	//Kapcsolat bontás
	bRobotSocketCloseEnable: BOOL := FALSE;
	RobotSocketClose: FB_SocketClose;
	
	bIsError : BOOL := FALSE;

END_VAR

RobotSocketOpen(
			sSrvNetId:= '', 
			sRemoteHost:= sRobotRemoteHost, 
			nRemotePort:= 2000, 
			bExecute:= bRobotSocketOpenEnable, 
			tTimeout:= T#45S, 
			bBusy=> bConnectBusy, 
			bError=> bConnectError, 
			nErrId=> nConnectErrId, 
			hSocket=> hRobotSocket);
			
RobotSocketSend(
		sSrvNetId:= '', 
		hSocket:= hRobotSocket, 
		cbLen:= uSendByteLen, 
		pSrc:= ADR(baSendByteArray), 
		bExecute:= bRobotSocketSendEnable, 
		tTimeout:= T#5S, 
		bBusy=> bSendBusy, 
		bError=> bSendError, 
		nErrId=> nSendErrId);
		
RobotSocketReceive(
	sSrvNetId:= '', 
	hSocket:= hRobotSocket, 
	cbLen:= 255, 
	pDest:= ADR(baReceivedByteArray), 
	bExecute:= bRobotSocketReceiveEnable, 
	tTimeout:= T#30S, 
	bBusy=> bReceiveBusy, 
	bError=> bReceiveError, 
	nErrId=> nReceiveErrId, 
	nRecBytes=> nRobotReceivedBytesNum);		
		
RobotSocketClose(
	sSrvNetId:= '', 
	hSocket:= hRobotSocket, 
	bExecute:= bRobotSocketCloseEnable, 
	tTimeout:= T#45S, 
	bBusy=> bCloseBusy, 
	bError=> bCloseError, 
	nErrId=> nCloseErrId);

//Kommunikáció nyitás
IF (bRobotCommOpenEnable = TRUE) AND (bRobotCommOpen = FALSE) AND (iState <= 0) THEN
	sRobotResult := '';	
	iState:=1;
ELSE
	bRobotCommOpenEnable := FALSE;
END_IF;

//Parancs küldés
IF (bRobotCommandSend = TRUE) AND (bRobotCommOpen=TRUE) AND(iState <= 0) THEN
	iState:=11;
ELSE
	bRobotCommandSend := FALSE;
END_IF;
//Kommunikáció zárás
IF (bRobotCommCloseEnable = TRUE) AND (bRobotCommOpen = TRUE) AND (iState < 31) THEN
	iState:=31;
ELSE
	bRobotCommCloseEnable := FALSE;
END_IF;




CASE iState OF
	
	1:	//Kommunikáció nyitás
		bRobotSocketOpenEnable:=TRUE;
		iState:=2;
	
	2:
		IF bConnectBusy = TRUE THEN
			iState:=3;
		END_IF
	3:
		IF bConnectBusy = FALSE THEN
			iState:=4;
		END_IF 
		
	4:
		IF bConnectError =FALSE THEN
			//Minden OK
			bRobotCommOpen:=TRUE;
		ELSE
			//HIBA
			bRobotCommOpen:=FALSE;	
		END_IF
		bRobotCommOpenEnable := FALSE;
		bRobotSocketOpenEnable:=FALSE;
		iState:=0;
		
		
	11: //Parancs küldés
		sRobotResult := '';
		nRobotErrId := 0;
		sLRobotCommand := sRobotCommand;
		sRobotSendData := sLRobotCommand;
		baSendByteArray := MAXSTRING_TO_BYTEARR(sRobotSendData);
		uSendByteLen := INT_TO_UDINT(LEN(sRobotSendData));
		MEMSET(ADR(baReceivedByteArray), 0, 256);
		
		iState:=12;
		
	12:
		bRobotSocketSendEnable:=TRUE;
		iState:=13;
		
	13:
		IF bSendBusy = TRUE THEN
			iState:=14;
		END_IF
	14:
		IF bSendBusy = FALSE THEN
			iState:=15;
		END_IF 
		
	15:
		IF bSendError =FALSE THEN
			//Minden OK
			bIsError:= FALSE;
			bRobotSocketReceiveEnable := FALSE;
			iState:=21;
		ELSE
			//HIBA
			bIsError:= TRUE;	
			iState:=0;
		END_IF
		bRobotCommandSend := FALSE;
		bRobotSocketSendEnable:=FALSE;
		
		sRobotCommand:='';		
		sLRobotCommand := '';

		
	21:	//Adatfogadás
		nRobotReceivedBytesNum:=0;
		bRobotSocketReceiveEnable := TRUE;
		iState:=22;
		
	22:
		IF bReceiveBusy = TRUE THEN
			iState:=23;
		END_IF
	23:
		IF bReceiveBusy = FALSE THEN
			iState:=24;
		END_IF 		
	24:
		IF bReceiveError =FALSE THEN
			//Minden OK
			bIsError:= FALSE;
			iState:=25;
		ELSE
			//HIBA
			bIsError:= TRUE;
			iState:=0;	
		END_IF
		bRobotSocketReceiveEnable:=FALSE;
		
	25:
		IF (nRobotReceivedBytesNum <>0) THEN
			sRobotReceived := BYTEARR_TO_MAXSTRING(baReceivedByteArray);
			IF sRobotReceived[0] = 16#30 THEN
				nRobotErrId:= 0;
			ELSE
				nRobotErrId:= 10000;
			END_IF
			GVL.stRobotStatusz:=f_GetRobotState(sRobotReceived);
			sRobotResult:=GVL.stRobotStatusz.sResult;
			iState:=0;
		ELSE
			iState:=21;
		END_IF
		

		
	31:	//Kommunikáció zárás
		bRobotSocketCloseEnable:=TRUE;
		iState:=32;
	
	32:
		IF bCloseBusy = TRUE THEN
			iState:=33;
		END_IF
	33:
		IF bCloseBusy = FALSE THEN
			bRobotSocketCloseEnable:=FALSE;
			iState:=34;
		END_IF 
		
	34:
		IF bCloseError =FALSE THEN
			//Minden OK
			bRobotCommOpen:=FALSE;
		ELSE
			//HIBA
			bRobotCommOpen:=FALSE;	//még át kell gondolni
		END_IF
		bRobotCommCloseEnable := FALSE;
		bRobotSocketCloseEnable:=FALSE;
		iState:=0;
	
END_CASE

END_PROGRAM

// ---- POUs/GENERAL/Helpers/f_GetRobotState.TcPOU
FUNCTION f_GetRobotState : ST_RobotState
VAR_INPUT
	sRobotValasz: STRING;
END_VAR
VAR
	sTemp: STRING;
	sRobotResult: STRING;
	sRobotInput: STRING;
	sRobotCoords: STRING;
	sX: STRING;
	sY: STRING;
	sZ: STRING;
	sU: STRING;
	sHand: STRING;
	nRobotInput: BYTE;
	iDelimiterPos: INT;
END_VAR

sTemp := DELETE(sRobotValasz,1,1);	// Első karakter (0/1) eltávolítása
sTemp := LEFT(sTemp,LEN(sTemp)-2);	// Utolsó két karakter ($R$N) eltávolítása
iDelimiterPos := FIND(sTemp,',');	// Első vessző helye
f_GetRobotState.sResult := LEFT(sTemp,iDelimiterPos-1);	// Vessző előtti szöveg
sTemp := RIGHT(sTemp,LEN(sTemp)-iDelimiterPos); // Vessző utáni szöveg
iDelimiterPos := FIND(sTemp,',');	// Második vessző helye
sRobotInput := LEFT(sTemp,iDelimiterPos-1);	// Vessző előtti szöveg
sTemp := RIGHT(sTemp,LEN(sTemp)-iDelimiterPos); // Vessző utáni szöveg			
iDelimiterPos := FIND(sTemp,',');	// Harmadik vessző helye
sX := LEFT(sTemp,iDelimiterPos-1);	// Vessző előtti szöveg
sTemp := RIGHT(sTemp,LEN(sTemp)-iDelimiterPos); // Vessző utáni szöveg			
iDelimiterPos := FIND(sTemp,',');	// Negyedik vessző helye
sY := LEFT(sTemp,iDelimiterPos-1);	// Vessző előtti szöveg
sTemp := RIGHT(sTemp,LEN(sTemp)-iDelimiterPos); // Vessző utáni szöveg			
iDelimiterPos := FIND(sTemp,',');	// Ötödik vessző helye
sZ := LEFT(sTemp,iDelimiterPos-1); // Vessző előtti szöveg
sTemp := RIGHT(sTemp,LEN(sTemp)-iDelimiterPos); // Vessző utáni szöveg			
iDelimiterPos := FIND(sTemp,',');	// Hatodik vessző helye
sU := LEFT(sTemp,iDelimiterPos-1); // Vessző előtti szöveg			
sHand := RIGHT(sTemp,LEN(sTemp)-iDelimiterPos);	// Vessző utáni szöveg
// nRobotInput bitekre bontása:
nRobotInput := STRING_TO_BYTE(sRobotInput);
f_GetRobotState.bVakuumSzippantoFent:=((nRobotInput AND 1) > 0);
f_GetRobotState.bVakuumSzippantoLent:=((nRobotInput AND 2) > 0);
f_GetRobotState.bCsipeszNyitva:=((nRobotInput AND 4) > 0);
f_GetRobotState.bCsipeszZarva:=((nRobotInput AND 8) > 0);
f_GetRobotState.bVakuumA:=((nRobotInput AND 16) > 0);
f_GetRobotState.bVakuumB:=((nRobotInput AND 32) > 0);
// Robot koordináták:
f_GetRobotState.rX:=STRING_TO_REAL(sX);
f_GetRobotState.rY:=STRING_TO_REAL(sY);
f_GetRobotState.rZ:=STRING_TO_REAL(sZ);
f_GetRobotState.rU:=STRING_TO_REAL(sU);
IF sHand='1' THEN
	sHand:='/R';
ELSIF sHand='2' THEN
	sHand:='/L';
ELSE
	sHand:='/?';
END_IF
f_GetRobotState.sHand:=sHand;

END_FUNCTION

// ---- POUs/JOZSI/Components/HAJLITOK.TcPOU
PROGRAM HAJLITOK
	VAR_INPUT
		s_InCommand : STRING := '';
		s_InCommandParam1 : STRING := '';
		s_InCommandParam2 : STRING := '';
		s_InCommandParam3 : STRING := '';
		s_InCommandParam4 : STRING := '';
		s_InCommandParam5 : STRING := '';
	END_VAR
	VAR_OUTPUT
		n_OutErrId: UINT;
	END_VAR
VAR
	bElohajlitoFelso AT %Q*: BOOL := FALSE;
	bElohajlitoAlso AT %Q*: BOOL := FALSE;
	bVeghajlitoFelso AT %Q*: BOOL := FALSE;
	bVeghajlitoAlso AT %Q*: BOOL := FALSE;
	bElohajlitoFelsoFent AT %I*: BOOL;
	bElohajlitoFelsoLent AT %I*: BOOL;
	bElohajlitoAlsoFent AT %I*: BOOL;
	bElohajlitoAlsoLent AT %I*: BOOL;
	bVeghajlitoFelsoFent AT %I*: BOOL;
	bVeghajlitoFelsoLent AT %I*: BOOL;
	bVeghajlitoAlsoFent AT %I*: BOOL;
	bVeghajlitoAlsoLent AT %I*: BOOL;
	iState : INT := 0;
	s_InLCommand : STRING := '';
	T_Ticker : TON;
	bTickerEnable : BOOL := FALSE;
	tTickerTime : TIME := T#300MS;
	bTickerQ : BOOL := FALSE;
END_VAR

IF HAJLITOK.s_InCommand <>'' AND s_InLCommand = '' THEN
	s_InLCommand := HAJLITOK.s_InCommand;
END_IF
IF s_InLCommand <> '' THEN
	IF iState = 0 AND s_InLCommand = 'ELOHAJLITAS' THEN
		iState := 1;
	END_IF
	IF iState = 0 AND s_InLCommand = 'VEGHAJLITAS' THEN
		iState := 51;
	END_IF
	CASE iState OF 
		1:
			IF (bElohajlitoFelsoFent = TRUE AND bElohajlitoFelsoLent = FALSE
				AND bElohajlitoAlsoFent = FALSE AND bElohajlitoAlsoLent = TRUE) THEN
				n_OutErrId := 0;
				iState := 2;
			ELSIF MAIN.bLevegoOK = FALSE THEN
				n_OutErrId := 5;
			ELSIF bElohajlitoFelsoFent = FALSE THEN
				n_OutErrId := 147;
			ELSIF bElohajlitoFelsoLent = TRUE THEN
				n_OutErrId := 146;
			ELSIF bElohajlitoAlsoFent = TRUE THEN
				n_OutErrId := 151;
			ELSIF bElohajlitoAlsoLent = FALSE THEN
				n_OutErrId := 149;
			END_IF
		2:	// Csak akkor menjen le, ha senki nem nyúlt be
			bElohajlitoFelso := GVL.bFenysorompoNTC;
			iState := 3;
		3:
			IF (bElohajlitoFelsoFent = FALSE AND bElohajlitoFelsoLent = TRUE
				AND bElohajlitoAlsoFent = FALSE AND bElohajlitoAlsoLent = TRUE) THEN
				n_OutErrId := 0;
				iState := 4;
			ELSE
				IF MAIN.bLevegoOK = FALSE THEN
					n_OutErrId := 5;
				ELSIF GVL.bFenysorompoNTC=FALSE THEN
					n_OutErrId := 31;
				ELSIF bElohajlitoFelsoFent = TRUE THEN
					n_OutErrId := 148;
				ELSIF bElohajlitoAlsoFent = TRUE THEN
					n_OutErrId := 152;
				ELSIF bElohajlitoAlsoLent = FALSE THEN
					n_OutErrId := 149;
				END_IF
				bElohajlitoFelso := GVL.bFenysorompoNTC;
			END_IF
		4:	// Csak akkor jöjjön fel, ha senki nem nyúlt be
			bElohajlitoAlso := GVL.bFenysorompoNTC;
			iState := 5;
		5:
			IF (bElohajlitoFelsoFent = FALSE AND bElohajlitoFelsoLent = TRUE
				AND bElohajlitoAlsoFent = TRUE AND bElohajlitoAlsoLent = FALSE) THEN
				n_OutErrId := 0;
				iState := 6;
			ELSE
				IF MAIN.bLevegoOK = FALSE THEN
					n_OutErrId := 5;
				ELSIF GVL.bFenysorompoNTC=FALSE THEN
					n_OutErrId := 31;
				ELSIF bElohajlitoFelsoFent = TRUE THEN
					n_OutErrId := 148;
				ELSIF bElohajlitoAlsoFent = TRUE THEN
					n_OutErrId := 152;
				ELSIF bElohajlitoAlsoLent = FALSE THEN
					n_OutErrId := 149;
				END_IF
				bElohajlitoAlso := GVL.bFenysorompoNTC;
			END_IF
		6:
			IF bTickerEnable = TRUE THEN
				bTickerEnable := FALSE;
			ELSE
				bTickerEnable := TRUE;
				iState := 7;
			END_IF
		7:
			IF bTickerQ = TRUE THEN
				bTickerEnable := FALSE;
				iState := 8;
			END_IF
		8:
			bElohajlitoAlso := FALSE;
			iState := 9;
		9:
			IF (bElohajlitoFelsoFent = FALSE AND bElohajlitoFelsoLent = TRUE
				AND bElohajlitoAlsoFent = FALSE AND bElohajlitoAlsoLent = TRUE) THEN
				n_OutErrId := 0;
				iState := 10;
			ELSIF MAIN.bLevegoOK = FALSE THEN
					n_OutErrId := 5;
			ELSIF bElohajlitoFelsoFent = TRUE THEN
				n_OutErrId := 148;
			ELSIF bElohajlitoFelsoLent = FALSE THEN
				n_OutErrId := 145;
			ELSIF bElohajlitoAlsoFent = TRUE THEN
				n_OutErrId := 152;
			ELSIF bElohajlitoAlsoLent = FALSE THEN
				n_OutErrId := 149;
			END_IF
		10:
			bElohajlitoFelso := FALSE;
			iState := 11;
		11:
			IF (bElohajlitoFelsoFent = TRUE AND bElohajlitoFelsoLent = FALSE
				AND bElohajlitoAlsoFent = FALSE AND bElohajlitoAlsoLent = TRUE) THEN
				iState := 0;
				n_OutErrId := 0;
			ELSIF MAIN.bLevegoOK = FALSE THEN
					n_OutErrId := 5;
			ELSIF bElohajlitoFelsoFent = FALSE THEN
					n_OutErrId := 147;
			ELSIF bElohajlitoFelsoLent = TRUE THEN
					n_OutErrId := 146;
			ELSIF bElohajlitoAlsoFent = TRUE THEN
					n_OutErrId := 152;
			ELSIF bElohajlitoAlsoLent = FALSE THEN
					n_OutErrId := 149;
			END_IF
			
		51:
			IF (bVeghajlitoFelsoFent = TRUE AND bVeghajlitoFelsoLent = FALSE
				AND bVeghajlitoAlsoFent = FALSE AND bVeghajlitoAlsoLent = TRUE) THEN
				n_OutErrId := 0;
				iState := 52;
			ELSIF MAIN.bLevegoOK = FALSE THEN
					n_OutErrId := 5;
			ELSIF bVeghajlitoFelsoFent = FALSE THEN
					n_OutErrId := 163;
			ELSIF bVeghajlitoFelsoLent = TRUE THEN
					n_OutErrId := 162;
			ELSIF bVeghajlitoAlsoFent = TRUE THEN
					n_OutErrId := 166;
			ELSIF bVeghajlitoAlsoLent = FALSE THEN
					n_OutErrId := 167;
			END_IF
		52:
			bVeghajlitoFelso := TRUE;
			iState := 53;
		53:
			IF (bVeghajlitoFelsoFent = FALSE AND bVeghajlitoFelsoLent = TRUE
				AND bVeghajlitoAlsoFent = FALSE AND bVeghajlitoAlsoLent = TRUE) THEN
				n_OutErrId := 0;
				iState := 54;
			ELSIF MAIN.bLevegoOK = FALSE THEN
					n_OutErrId := 5;
			ELSIF bVeghajlitoFelsoFent = TRUE THEN
					n_OutErrId := 164;
			ELSIF bVeghajlitoFelsoLent = FALSE THEN
					n_OutErrId := 161;
			ELSIF bVeghajlitoAlsoFent = TRUE THEN
					n_OutErrId := 166;
			ELSIF bVeghajlitoAlsoLent = FALSE THEN
					n_OutErrId := 167;
			END_IF
		54:
			bVeghajlitoAlso := TRUE;
			iState := 55;
		55:
			IF (bVeghajlitoFelsoFent = FALSE AND bVeghajlitoFelsoLent = TRUE
				AND bVeghajlitoAlsoFent = TRUE AND bVeghajlitoAlsoLent = FALSE) THEN
				n_OutErrId := 0;
				iState := 56;
			ELSIF MAIN.bLevegoOK = FALSE THEN
					n_OutErrId := 5;
			ELSIF bVeghajlitoFelsoFent = TRUE THEN
					n_OutErrId := 164;
			ELSIF bVeghajlitoFelsoLent = FALSE THEN
					n_OutErrId := 161;
			ELSIF bVeghajlitoAlsoFent = FALSE THEN
					n_OutErrId := 165;
			ELSIF bVeghajlitoAlsoLent = TRUE THEN
					n_OutErrId := 168;
			END_IF
		56:
			IF bTickerEnable = TRUE THEN
				bTickerEnable := FALSE;
			ELSE
				bTickerEnable := TRUE;
				iState := 57;
			END_IF
		57:
			IF bTickerQ = TRUE THEN
				bTickerEnable := FALSE;
				iState := 58;
			END_IF
		58:
			bVeghajlitoAlso := FALSE;
			iState := 59;
		59:
			IF (bVeghajlitoFelsoFent = FALSE AND bVeghajlitoFelsoLent = TRUE
				AND bVeghajlitoAlsoFent = FALSE AND bVeghajlitoAlsoLent = TRUE) THEN
				n_OutErrId := 0;
				iState := 60;
			ELSIF MAIN.bLevegoOK = FALSE THEN
				n_OutErrId := 5;
			ELSIF bVeghajlitoFelsoFent = TRUE THEN
				n_OutErrId := 164;
			ELSIF bVeghajlitoFelsoLent = FALSE THEN
				n_OutErrId := 161;
			ELSIF bVeghajlitoAlsoFent = TRUE THEN
				n_OutErrId := 166;
			ELSIF bVeghajlitoAlsoLent = FALSE THEN
				n_OutErrId := 167;
			END_IF
		60:
			bVeghajlitoFelso := FALSE;
			iState := 61;
		61:
			IF (bVeghajlitoFelsoFent = TRUE AND bVeghajlitoFelsoLent = FALSE
				AND bVeghajlitoAlsoFent = FALSE AND bVeghajlitoAlsoLent = TRUE) THEN
				iState := 0;
				n_OutErrId := 0;
			ELSIF MAIN.bLevegoOK = FALSE THEN
				n_OutErrId := 5;
			ELSIF bVeghajlitoFelsoFent = FALSE THEN
				n_OutErrId := 163;
			ELSIF bVeghajlitoFelsoLent = TRUE THEN
				n_OutErrId := 162;
			ELSIF bVeghajlitoAlsoFent = TRUE THEN
				n_OutErrId := 166;
			ELSIF bVeghajlitoAlsoLent = FALSE THEN
				n_OutErrId := 167;
			END_IF
			
	END_CASE
	IF iState = 0 THEN
		HAJLITOK.s_InCommand := '';
		s_InLCommand := '';
	END_IF
END_IF

T_Ticker(IN:= bTickerEnable, PT:= tTickerTime, Q=> bTickerQ, ET=> );

END_PROGRAM

// ---- POUs/PISTI/Components/PISTITENGELY.TcPOU
PROGRAM PISTITENGELY
VAR
	PistiHome: MC_Home;
	bPistiHomeEnable: BOOL := FALSE;
	bAxisBusy : BOOL := FALSE;
	bAxisActive: BOOL := FALSE;
	bAxisAborted: BOOL := FALSE;
	bAxisError: BOOL := FALSE;
	nAxisErrorID: UDINT;
	bAxisStopDone: BOOL := FALSE;
	bPistiHomeSwitch AT %I*: BOOL;
	fbPistiTengelyStop: MC_Stop;
	fbPistitengelyServo: MC_Power;
	bPistiPosSwitch : BOOL := TRUE;
	bPistiTengelySzabad : BOOL;
	bOperational AT %I*: BOOL;
	bHomeReady : BOOL := FALSE;
	nAxisStatus AT %I*: UINT;
	bAxisReady : BOOL;
	bAxisOn : BOOL;
	
	//HOME
	bAxisHomeDone: BOOL;
	bAxisHomeBusy: BOOL;
	bAxisHomeActive: BOOL;
	bAxisHomeAborted: BOOL;
	bAxisHomeError: BOOL;
	nAxisHomeErrorID: UDINT;
	
	//MOVE
	bAxisMoveDone: BOOL;
	bAxisMoveBusy: BOOL;
	bAxisMoveActive: BOOL;
	bAxisMoveAborted: BOOL;
	bAxisMoveError: BOOL;
	nAxisMoveErrorID: UDINT;
	
	//COMMAND
	bAxisCommandDone: BOOL;
	bAxisCommandBusy: BOOL;
	bAxisCommandActive: BOOL;
	bAxisCommandAborted: BOOL;
	bAxisCommandError: BOOL;
	nAxisCommandErrorID: UDINT;
	
	
	fbPistitengelyJOG: MC_Jog;
	bPistiJOGPlus : BOOL := FALSE;
	bPistiJOGMinus : BOOL := FALSE;
	fbPistitengelyReset: MC_Reset;
	bPistiReset: BOOL;
	nPistiErrorCode AT %I*: UDINT;
	lrPistiActPos AT %I*: LREAL;
	fbPistiMoveAbolute: MC_MoveAbsolute;
	
	//Pozicioknak
//	lrSzervizbox : LREAL := -5;
//	lrHegesztoPosition1 : LREAL := -398.3;
//	lrHegesztoPosition2 : LREAL := -404.3;
//	lrRobotpakolasPosition : LREAL := -617.8125;
//	lrKodolvasasPosition: LREAL := -841.54;
//	lrKappePosition : LREAL := -837.227;
//	lrVegmeroPosition : LREAL := -1054.776;
	bPistiTengelySzabad_TON: TON;
END_VAR
VAR_INPUT
	lrPistiPosition : LREAL := 0;
	sPistiAxisCommand: STRING := '';
END_VAR
VAR_OUTPUT
	n_OutErrId: UINT;
END_VAR

//bPistiTengelySzabad := GVL.bTempPistiInputs1[3] AND GVL.bTempPistiInputs2[6]
bPistiTengelySzabad := GVL.bHegeszto3Fent AND GVL.bKappepresFent
						AND VEGMERO.bMerotukBent AND (HIMBA.bHimba_hatul AND NOT HIMBA.bHimba_elol) AND bOperational
//						AND ((GVL.stRobotStatusz.rX<-1.0) OR (GVL.stRobotStatusz.rZ>-111.0))
						AND f_RobotPtTengelytolTavol()
						AND (GVL.bFenysorompoPt
							OR (sPistiAxisCommand='HOME')
							OR (PISTITENGELY.lrPistiActPos>-10)
							OR (PISTITENGELY.lrPistiActPos<-500))
						AND NOT GVL.bBiztonsagiFold AND GVL.bBiztonsagiTap;
bPistiTengelySzabad_TON(IN:=bPistiTengelySzabad, PT:=T#100MS);
IF bPistiTengelySzabad_TON.Q=FALSE THEN
	IF MAIN.bLevegoOK=FALSE THEN
		n_OutErrId:=5;
	ELSIF GVL.bHegeszto3Fent=FALSE THEN
		n_OutErrId:=71;
	ELSIF GVL.bKappepresFent=FALSE THEN
		n_OutErrId:=109;
	ELSIF VEGMERO.bMerotukBent=FALSE THEN
		n_OutErrId:=87;
	ELSIF HIMBA.bHimba_hatul=FALSE OR HIMBA.bHimba_elol=TRUE THEN
		n_OutErrId:=339;
	ELSIF bOperational=FALSE THEN
		n_OutErrId:=195;
//	ELSIF NOT ((GVL.stRobotStatusz.rX<-1.0) OR (GVL.stRobotStatusz.rZ>-111.0)) THEN
	ELSIF NOT f_RobotPtTengelytolTavol() THEN
		n_OutErrId:=302;
	ELSIF (GVL.bFenysorompoPt=FALSE) THEN
		n_OutErrId:=29;
	ELSIF GVL.bBiztonsagiFold=TRUE THEN
		n_OutErrId:=42;
	ELSIF GVL.bBiztonsagiTap=FALSE THEN
		n_OutErrId:=43;
	END_IF
ELSE
	n_OutErrId := 0;
END_IF
bAxisReady:=nAxisStatus MOD 2 = 1;
bAxisOn:=nAxisStatus/2 MOD 2 = 1;
fbPistiTengelyStop(
	Axis:= GVL.axisPistiTengely, 
	Execute:= (NOT((GVL.bPistiPosSwitch OR sPistiAxisCommand='HOME') AND GVL.bPistiNegSwitch AND bPistiTengelySzabad_TON.Q)
				OR sPistiAxisCommand='STOP'), 
	Deceleration:= , 
	Jerk:= , 
	Options:= , 
	Done=> PISTITENGELY.bAxisStopDone, 
	Busy=> bAxisBusy, 
	Active=> bAxisActive, 
	CommandAborted=> bAxisAborted, 
	Error=> bAxisError, 
	ErrorID=> nAxisErrorID);
IF (sPistiAxisCommand='STOP') AND PISTITENGELY.bAxisStopDone AND NOT bAxisError THEN
	sPistiAxisCommand := '';
END_IF
IF NOT(GVL.bPistiPosSwitch OR sPistiAxisCommand='HOME') OR NOT(GVL.bPistiNegSwitch) THEN
	GVL.bPistiServo := FALSE;
	sPistiAxisCommand:='';
END_IF
fbPistitengelyServo(
	Axis:= GVL.axisPistiTengely, 
	Enable:= GVL.bPistiServo, 
	Enable_Positive:= (GVL.bPistiPosSwitch OR sPistiAxisCommand='HOME'), 
	Enable_Negative:= GVL.bPistiNegSwitch, 
	Override:= 100, 
	BufferMode:= , 
	Options:= , 
	Status=> , 
	Busy=> , 
	Active=> , 
	Error=> , 
	ErrorID=> );
	
	//Home
PistiHome(
	Axis:= GVL.axisPistiTengely, 
	Execute:= sPistiAxisCommand='HOME' AND bPistiTengelySzabad_TON.Q, 
	Position:= DEFAULT_HOME_POSITION, 
	HomingMode:= MC_DefaultHoming, 
	BufferMode:= , 
	Options:= , 
	bCalibrationCam:= NOT(bPistiHomeSwitch), 
	Done=> bAxisHomeDone, 
	Busy=> bAxisHomeBusy, 
	Active=> bAxisHomeActive, 
	CommandAborted=> bAxisHomeAborted, 
	Error=> bAxisHomeError, 
	ErrorID=> nAxisHomeErrorID);
	//Lefutás ellenőrzése
IF (bAxisHomeDone AND NOT(bAxisHomeBusy OR bAxisHomeActive OR bAxisHomeAborted OR bAxisHomeError)) THEN
	lrPistiPosition:=GVL.lrPtSzervizbox;
	sPistiAxisCommand := 'MOVE';
	bHomeReady:=TRUE;
END_IF
	
	//Move
fbPistiMoveAbolute(
	Axis:= GVL.axisPistiTengely, 
	Execute:= sPistiAxisCommand='MOVE' AND bPistiTengelySzabad_TON.Q AND bHomeReady, 
	Position:= lrPistiPosition, // -1060...0
	Velocity:= 800, 
	Acceleration:= 0, 
	Deceleration:= 0, 
	Jerk:= 0, 
	BufferMode:= , 
	Options:= , 
	Done=> bAxisMoveDone, 
	Busy=> bAxisMoveBusy, 
	Active=> bAxisMoveActive, 
	CommandAborted=> bAxisMoveAborted, 
	Error=> bAxisMoveError, 
	ErrorID=> nAxisMoveErrorID);
	//Lefutás ellenőrzése
IF (bAxisMoveDone AND NOT(bAxisMoveBusy OR bAxisMoveActive OR bAxisMoveAborted OR bAxisMoveError)) THEN
	sPistiAxisCommand := '';
END_IF
	
	//JOG
	fbPistitengelyJOG(
	Axis:= GVL.axisPistiTengely, 
	JogForward:= bPistiJOGPlus AND bPistiTengelySzabad_TON.Q, 
	JogBackwards:= bPistiJOGMinus AND bPistiTengelySzabad_TON.Q, 
	Mode:= MC_JOGMODE_STANDARD_SLOW , 
	Position:= , 
	Velocity:= 100, 
	Acceleration:= 0, 
	Deceleration:= 0, 
	Jerk:= 0, 
	Done=> bAxisCommandDone, 
	Busy=> bAxisCommandBusy, 
	Active=> bAxisCommandActive, 
	CommandAborted=> bAxisCommandAborted, 
	Error=> bAxisCommandError, 
	ErrorID=> nAxisCommandErrorID);
	
	//RESET ERROR
	fbPistitengelyReset(
	Axis:= GVL.axisPistiTengely, 
	Execute:= bPistiReset, 
	Done=> bAxisCommandDone, 
	Busy=> bAxisCommandBusy, 
	Error=> bAxisCommandError, 
	ErrorID=> nAxisCommandErrorID);
	
	//Ha nem szabad futtatni
//	IF(NOT(bPistiTengelySzabad)) THEN
//		sPistiAxisCommand:='!INTERRUPTED';
//	END_IF

END_PROGRAM

// ---- POUs/PISTI/Components/HIMBA.TcPOU
PROGRAM HIMBA
VAR_INPUT
	s_InCommand : STRING := '';
	s_InCommandParam1 : STRING := '';
	s_InCommandParam2 : STRING := '';
	s_InCommandParam3 : STRING := '';
	s_InCommandParam4 : STRING := '';
	s_InCommandParam5 : STRING := '';
END_VAR
VAR_OUTPUT
	n_OutErrId: UINT;
END_VAR
VAR
	bHimba_hatul AT %I*: BOOL; //6
	bHimba_elol AT %I*: BOOL; //7
	bHimba_szenzor AT %I*: BOOL; //Bemenetek2 10
	bHimba AT %Q*: BOOL := 0; //Szelep11
	iState: INT;
	WAIT: TON;
	bStartWait: BOOL := FALSE;
	bIdoLejart: BOOL := FALSE;
	tDelay: TIME := T#2000MS;
END_VAR

IF (iState=0) AND (HIMBA.s_InCommand='START') THEN
	iState:=1;
ELSIF (iState<20) AND (HIMBA.s_InCommand='RESET') THEN
	iState:=20;
END_IF

	IF iState<>0 THEN
		CASE iState OF
		// Himba kitolása
		1:	GVL.bHimbaOK:=FALSE;
			HIMBA.bHimba:=TRUE;
			iState:=2;
		// Ha megérkezett a Himba, várunk a megnyugvásra
		2:	IF (HIMBA.bHimba_elol=TRUE) AND (HIMBA.bHimba_hatul=FALSE) THEN
				tDelay:=T#600MS;
				bStartWait:=TRUE;
				n_OutErrId:=0;
				iState:=3;
			ELSE
				n_OutErrId:=338;
			END_IF
		// Ha lejárt a várakozási idő kiértékeljük az érzékelő jelét
		3:	IF (bIdoLejart=TRUE) THEN
				bStartWait:=FALSE;
				IF (HIMBA.bHimba_szenzor=TRUE) THEN
					GVL.bHimbaOK:=TRUE;
				ELSE
					GVL.bHimbaOK:=FALSE;
				END_IF
				iState:=4;
			END_IF
		// Himba visszahúzása
		4:	HIMBA.bHimba:=FALSE;
			iState:=5;
		// Ha visszatért a himba, várunk a megnyugvásra
		5: IF (HIMBA.bHimba_hatul=TRUE) AND (HIMBA.bHimba_elol=FALSE) THEN
				tDelay:=T#300MS;
				bStartWait:=TRUE;
				n_OutErrId:=0;
				iState:=6;
			ELSE
				n_OutErrId:=339;
			END_IF
		// Ha lejárt az idő, vége a folyamatnak
		6:	IF (bIdoLejart=TRUE) THEN
				bStartWait:=FALSE;
				iState:=0;
				HIMBA.s_InCommand:='';
			END_IF

		// Reset: húzza vissza a himbát!
		20:	bStartWait:=FALSE;
			GVL.bHimbaOK:=FALSE;
			HIMBA.bHimba:=FALSE;
			iState:=21;				
		// Ha visszatért a himba, várunk a megnyugvásra
		21:	IF (HIMBA.bHimba_hatul=TRUE) AND (HIMBA.bHimba_elol=FALSE) THEN
				tDelay:=T#300MS;
				bStartWait:=TRUE;
				n_OutErrId:=0;
				iState:=22;
			ELSE
				n_OutErrId:=339;
			END_IF
		// Ha lejárt az idő, vége a folyamatnak
		22:	IF (bIdoLejart=TRUE) THEN
				bStartWait:=FALSE;
				iState:=0;
				HIMBA.s_InCommand:='';
			END_IF
		END_CASE
	END_IF	

WAIT(IN:=bStartWait,PT:=tDelay,Q=>bIdoLejart,ET=>);

END_PROGRAM

// ---- POUs/GENERAL/Helpers/f_RobotPtTengelytolTavol.TcPOU
FUNCTION f_RobotPtTengelytolTavol : BOOL

f_RobotPtTengelytolTavol:=(GVL.stRobotStatusz.rX<-1.0) OR (GVL.stRobotStatusz.rZ>-111.0);

END_FUNCTION

// ---- POUs/PISTI/Components/KAPPE.TcPOU
PROGRAM KAPPE
VAR_INPUT
	s_InCommand : STRING := '';
	s_InCommandParam1 : STRING := '';
	s_InCommandParam2 : STRING := '';
	s_InCommandParam3 : STRING := '';
	s_InCommandParam4 : STRING := '';
	s_InCommandParam5 : STRING := '';
END_VAR
VAR_OUTPUT
	n_OutErrId: UINT;
END_VAR
VAR
	bKappeFelLe AT %Q*: BOOL := 0;
	bKappeBalFelLe AT %Q*: BOOL := 0;
	bKappeJobbFelLe AT %Q*: BOOL := 0;
	bKappeNincsLegalul AT %I*: BOOL;
	bKappeFent AT %I*: BOOL;
	bKappeBalFent AT %I*: BOOL;
	bKappeBalLent AT %I*: BOOL;
	bKappeJobbFent AT %I*: BOOL;
	bKappeJobbLent AT %I*: BOOL;
	iState: INT;
	WAIT: TON;
	bStartWait: BOOL := FALSE;
	bIdoLejart: BOOL := FALSE;
	tDelay: TIME := T#2000MS;
END_VAR

IF (iState=0) AND (KAPPE.s_InCommand='START') THEN
	iState:=1;
ELSIF (iState<20) AND (KAPPE.s_InCommand='RESET') THEN
	iState:=20;
END_IF
	IF iState<>0 THEN
		CASE iState OF
		// Kappe fej leeresztése
		1:	KAPPE.bKappeFelLe:=TRUE;
			iState:=2;
		// Ha leérkezett a Kappe fej, akkor várakozik a nyugvópontra
		2:	IF (GVL.bKappepresNincsLegalul=FALSE) THEN
				tDelay:=T#200MS;
				bStartWait:=TRUE;
				n_OutErrId := 0;
				iState:=3;
			ELSE
				IF MAIN.bLevegoOK=FALSE THEN
					n_OutErrId:=5;
				ELSE
					n_OutErrId:=94;
				END_IF
			END_IF
		// Ha lejárt a várakozási idő és a kappézó ujjak ki vannak nyitva,
		// akkor zárja be az ujjakat!
		3:	IF (bIdoLejart=TRUE) AND (KAPPE.bKappeBalFent=TRUE) 
				AND (KAPPE.bKappeBalLent=FALSE) AND (KAPPE.bKappeJobbFent=TRUE)
				AND (KAPPE.bKappeJobbLent=FALSE) THEN
				bStartWait:=FALSE;
				KAPPE.bKappeBalFelLe:=TRUE;
				KAPPE.bKappeJobbFelLe:=TRUE;
				n_OutErrId := 0;
				iState:=4;
			ELSIF MAIN.bLevegoOK=FALSE THEN
				n_OutErrId:=5;
			ELSIF (KAPPE.bKappeBalFent=FALSE) THEN
				n_OutErrId:=101;
			ELSIF (KAPPE.bKappeBalLent=TRUE) THEN
				n_OutErrId:=104;
			ELSIF (KAPPE.bKappeJobbFent=FALSE) THEN
				n_OutErrId:=99;
			ELSIF (KAPPE.bKappeJobbLent=TRUE) THEN
				n_OutErrId:=98;
			END_IF
		// Ha megnyomta a Kappét, várjon egy kicsit!
		4:	IF (KAPPE.bKappeBalFent=FALSE) AND (KAPPE.bKappeBalLent=TRUE)
				AND (KAPPE.bKappeJobbFent=FALSE) AND (KAPPE.bKappeJobbLent=TRUE) THEN
				tDelay:=T#1000MS;
				bStartWait:=TRUE;
				n_OutErrId := 0;
				iState:=5;
			ELSIF MAIN.bLevegoOK=FALSE THEN
				n_OutErrId:=5;
			ELSIF (KAPPE.bKappeBalFent=TRUE) THEN
				n_OutErrId:=102;
			ELSIF (KAPPE.bKappeBalLent=FALSE) THEN
				n_OutErrId:=103;
			ELSIF (KAPPE.bKappeJobbFent=TRUE) THEN
				n_OutErrId:=100;
			ELSIF (KAPPE.bKappeJobbLent=FALSE) THEN
				n_OutErrId:=97;
			END_IF
		// A várakozás után nyissa ki a kappézó ujjakat!
		5:	IF (bIdoLejart=TRUE) THEN
				bStartWait:=FALSE;
				KAPPE.bKappeBalFelLe:=FALSE;
				KAPPE.bKappeJobbFelLe:=FALSE;
				iState:=6;				
			END_IF
		// Ha kinyíltak a kappézó ujjak, akkor Kappe fej fel
		6:	IF (KAPPE.bKappeBalFent=TRUE) AND (KAPPE.bKappeBalLent=FALSE)
				AND (KAPPE.bKappeJobbFent=TRUE) AND (KAPPE.bKappeJobbLent=FALSE) THEN
				KAPPE.bKappeFelLe:=FALSE;
				tDelay:=T#2000MS;
				bStartWait:=TRUE;
				n_OutErrId := 0;
				iState:=7;
			ELSIF MAIN.bLevegoOK=FALSE THEN
				n_OutErrId:=5;
			ELSIF (KAPPE.bKappeBalFent=FALSE) THEN
				n_OutErrId:=101;
			ELSIF (KAPPE.bKappeBalLent=TRUE) THEN
				n_OutErrId:=104;
			ELSIF (KAPPE.bKappeJobbFent=FALSE) THEN
				n_OutErrId:=99;
			ELSIF (KAPPE.bKappeJobbLent=TRUE) THEN				
				n_OutErrId:=98;
			END_IF
		// Ha felemelkedett a Kappe fej, akkor vége a folyamatnak
		7:	IF (GVL.bKappePresFent=TRUE) THEN
				bStartWait:=FALSE;				
				n_OutErrId:=0;
				iState:=0;
				KAPPE.s_InCommand:='';
			ELSIF MAIN.bLevegoOK=FALSE THEN
				n_OutErrId:=5;
			ELSIF (GVL.bKappePresFent=FALSE) THEN
				n_OutErrId:=205;
			END_IF
		// Reset: nyissa ki a kappézó ujjakat!
		20:	bStartWait:=FALSE;
			KAPPE.bKappeBalFelLe:=FALSE;
			KAPPE.bKappeJobbFelLe:=FALSE;
			iState:=21;				
		// Ha kinyíltak a kappézó ujjak, akkor Kappe fej fel
		21:	IF (KAPPE.bKappeBalFent=TRUE) AND (KAPPE.bKappeBalLent=FALSE)
				AND (KAPPE.bKappeJobbFent=TRUE) AND (KAPPE.bKappeJobbLent=FALSE) THEN
				KAPPE.bKappeFelLe:=FALSE;
				tDelay:=T#2000MS;
				bStartWait:=TRUE;
				n_OutErrId := 0;
				iState:=22;
			ELSIF MAIN.bLevegoOK=FALSE THEN
				n_OutErrId:=5;
			ELSIF (KAPPE.bKappeBalFent=FALSE) THEN
				n_OutErrId:=101;
			ELSIF (KAPPE.bKappeBalLent=TRUE) THEN
				n_OutErrId:=104;
			ELSIF (KAPPE.bKappeJobbFent=FALSE) THEN
				n_OutErrId:=99;
			ELSIF (KAPPE.bKappeJobbLent=TRUE) THEN				
				n_OutErrId:=98;
			END_IF
		// Ha felemelkedett a Kappe fej, akkor vége a folyamatnak
		22:	IF (GVL.bKappePresFent=TRUE) THEN
				bStartWait:=FALSE;				
				n_OutErrId:=0;
				iState:=0;
				KAPPE.s_InCommand:='';
			ELSIF MAIN.bLevegoOK=FALSE THEN
				n_OutErrId:=5;
			ELSIF (GVL.bKappePresFent=FALSE) THEN
				n_OutErrId:=205;
			END_IF
		END_CASE
	END_IF	
WAIT(IN:=bStartWait,PT:=tDelay,Q=>bIdoLejart,ET=>);

END_PROGRAM

// ---- POUs/GENERAL/Components/TERMEKVALTAS.TcPOU
PROGRAM TERMEKVALTAS
VAR_INPUT
	iState: INT := 1;
	bStart: BOOL := FALSE;
END_VAR
VAR_OUTPUT
	bOK: BOOL := FALSE;
	bBusy: BOOL := FALSE;
END_VAR

CASE iState OF
	1:
		IF (GVL.iPreviousSelectedProductType<>GVL.iSelectedProductType) OR
			(bStart=TRUE) THEN
			bOK:=FALSE;
			bBusy:=TRUE;
			iState:=2;
			GVL.iCurrentProductType:=-3; // Kérje az etalonokat!
		END_IF
	2:
		IF NOT(GVL.iSelectedProductType=8) THEN
			IF(GVL.iSelectedProductType<8) THEN
				Laser.s_InCommand:='SETJOB_637';
			ELSE
				CASE GVL.iSelectedProductType OF
					9, 11, 13, 15: Laser.s_InCommand:='SETJOB_745900';
					10, 12, 14, 16: Laser.s_InCommand:='SETJOB_745910';
				END_CASE
(*			ELSIF GVL.iSelectedProductType=9 THEN
				Laser.s_InCommand:='SETJOB_745900';
			ELSIF GVL.iSelectedProductType=10 THEN
				Laser.s_InCommand:='SETJOB_745910';*)
			END_IF;
			GVL.bKameraBe := TRUE;
			GVL.bHajlitasBe := TRUE;
			GVL.bHegesztes1Be := TRUE;
			GVL.bHegesztes2Be := TRUE;
			GVL.bHegesztes3Be := TRUE;
			GVL.bHegesztes4Be := TRUE;
			GVL.bHegesztes5Be := TRUE;
			GVL.bKameraVegBe := FALSE;
			GVL.bHegesztes6Be := TRUE;
			GVL.bHegesztes7Be := TRUE;
			GVL.bPtKameraBe := TRUE;
			GVL.bRobotKappeBe := FALSE;
			GVL.bKappeBe := TRUE;
			GVL.bMeresBe := TRUE;
			IF (GVL.iSelectedProductType>8) THEN
				GVL.bHimbaBe := TRUE;
			ELSE
				GVL.bHimbaBe := FALSE;
			END_IF
			GVL.bJelolesBe := TRUE;	
			iState:=3;
		ELSIF GVL.iSelectedProductType=8 THEN
			Laser.s_InCommand:='SETJOB_521';
			GVL.bKameraBe := FALSE;
			GVL.bHajlitasBe := FALSE;
			GVL.bHegesztes1Be := FALSE;
			GVL.bHegesztes2Be := FALSE;
			GVL.bHegesztes3Be := FALSE;
			GVL.bHegesztes4Be := FALSE;
			GVL.bHegesztes5Be := FALSE;
			GVL.bKameraVegBe := FALSE;
			GVL.bHegesztes6Be := FALSE;
			GVL.bHegesztes7Be := FALSE;
			GVL.bPtKameraBe := FALSE;
			GVL.bRobotKappeBe := FALSE;
			GVL.bKappeBe := FALSE;
			GVL.bMeresBe := FALSE;
			GVL.bHimbaBe := FALSE;
			GVL.bJelolesBe := TRUE;	
			iState:=4;
		ELSE
			iState:=1;
			GVL.iSelectedProductType:=GVL.iPreviousSelectedProductType;
			bOK:=FALSE;
			bBusy:=FALSE;
		END_IF
	3:
		IF Laser.s_InCommand='' THEN
			Laser.s_InCommand:='SETTYPE';
			iState:=4;
		END_IF
	4:
		IF Laser.s_InCommand='' THEN
			iState:=1;
			bOK:=TRUE;
			bBusy:=FALSE;
			bStart:=FALSE;
			GVL.iPreviousSelectedProductType:=GVL.iSelectedProductType;
		ELSIF Laser.s_InCommand<>'SETTYPE' THEN
			iState:=1;
			bOK:=FALSE;
			bBusy:=FALSE;
			bStart:=FALSE;
			GVL.iPreviousSelectedProductType:=GVL.iSelectedProductType;
		END_IF	
END_CASE

END_PROGRAM

// ---- POUs/PISTI/Components/ZEBRASCANNER.TcPOU
PROGRAM ZEBRASCANNER
VAR
	iState: INT := 0;
	// I/O variables for a PC COM PORT
	InputBuffer AT %I*: PcComInData;
	OutputBuffer AT %Q*: PcComOutData;
	TxBufferPcCom: COMbuffer;
	RxBufferPcCom: COMbuffer;

	// Serial line control for virtual COM port
	fbPCComCtrl: SerialLineControlADS;
	bConnect: BOOL := TRUE;
//	stSerialCfg: ComSerialConfig := (ComPort := 5, DTR := COMDTRCTRL_T.DTR_CTRL_DISABLE, RTS := COMRTSCTRL_T.RTS_CTRL_ENABLE);
	stSerialCfg: ComSerialConfig := (ComPort := 7, Baudrate:=115200, Parity:=PARITY_EVEN, DTR := COMDTRCTRL_T.DTR_CTRL_DISABLE, RTS := COMRTSCTRL_T.RTS_CTRL_ENABLE);
	stSerialCfgZebra: ComSerialConfig := (ComPort := 5, DTR := COMDTRCTRL_T.DTR_CTRL_DISABLE, RTS := COMRTSCTRL_T.RTS_CTRL_ENABLE);
	stSerialCfgKeyence: ComSerialConfig := (ComPort := 7, Baudrate:=115200, Parity:=PARITY_EVEN, DTR := COMDTRCTRL_T.DTR_CTRL_DISABLE, RTS := COMRTSCTRL_T.RTS_CTRL_ENABLE);
	bPortOpened: BOOL;
	bPcComCtrlError: BOOL;
	ePcComCtrlErrorId: UDINT;
	bPCComCtrlBusy: BOOL;
	uiTxBufferCount: UDINT;
	uiRxBufferCount: UDINT;
	
//	fbPCComCtrl2: SerialLineControl;
	
	// Receiving
	ZebraReceiveString: ReceiveString;
	bReset: BOOL;
	sReceivedString: STRING;
	bStringReceived: BOOL;
	bBusy: BOOL;
	cetError: ComError_t;
	bRxTimeout: BOOL;
	
	// Sending
	ZebraSendString: SendString;	
	sStringToSend: STRING;
	bSendBusy: BOOL;
	eSendError: ComError_t;
	sStartScanning: STRING := '$04$E4$04$00$00$14';
	iSendDataLength: UDINT := 6;
	
	// Sending bytes
	nSentBytes: DINT;
	ZebraSendData: SendData;
	
	// Receiving bytes
	nReceivedBytes: DINT;
	baReceivedBytes: ARRAY[0..255] OF BYTE;
	ZebraReceiveBytes: ReceiveByte;
	ReceiveString255: ReceiveString255;
	ClearComBuffer: ClearComBuffer;
	sExpectedString: T_MaxString;
	
	GetTime: NT_GetTime;
	bStartGetTime: BOOL;
	bGetTimeBusy: BOOL;
	bGetTimeError: BOOL;
	nGetTimeError: UDINT;
	sYear: STRING;
	sMonth: STRING;
	sDay: STRING;
	tstDateTime: TIMESTRUCT;
	sTypeCode: STRING;
	Timer: TON;
	bStart: BOOL;
	tTimeOut: TIME := T#3S;
	bTimeOut: BOOL;
	tElapsedTime: TIME;
	bKeyence: BOOL;
	iInd: INT;
END_VAR

VAR_INPUT
	bStartSend: BOOL;	
END_VAR

VAR_OUTPUT
	sReceivedString255: T_MaxString;
	nReceivedStringLength: DINT;
	bReadReady: BOOL := FALSE;	
END_VAR

(*VAR_IN_OUT
	sExpectedString: T_MaxString;
END_VAR*)

VAR CONSTANT
	baStartScanning: ARRAY[0..5] OF BYTE := [16#4, 16#E4, 16#4, 16#0, 16#FF, 16#14];
	baStartScanningKeyence: ARRAY[0..3] OF BYTE := [16#4C, 16#4F, 16#4E, 16#0D];
END_VAR

fbPCComCtrl(
	Connect:=bConnect,
	SerialCfg:=stSerialCfg,
	NetId:='',
	Timeout:=T#2s,
	PortOpened=>bPortOpened,
	Error=>bPCComCtrlError,
	ErrorId=>ePCComCtrlErrorId,
	Busy=>bPCComCtrlBusy,
	TxBufCount=>uiTxBufferCount,
	RxBufCount=>uiRxBufferCount,
	TxBuffer:=TxBufferPcCom,
	RxBuffer:=RxBufferPcCom);

REPEAT
	ZebraReceiveBytes(Rxbuffer:=RxBufferPcCom);
	IF ZebraReceiveBytes.ByteReceived THEN
		IF nReceivedBytes=0 THEN
			FOR nReceivedBytes:=0 TO 255 DO
				baReceivedBytes[nReceivedBytes]:=0;
			END_FOR
			nReceivedBytes:=0;
		END_IF
		baReceivedBytes[nReceivedBytes]:=ZebraReceiveBytes.ReceivedByte;
		nReceivedBytes:=nReceivedBytes+1;
	END_IF
UNTIL NOT ZebraReceiveBytes.ByteReceived
END_REPEAT;

(*REPEAT
	ReceiveString255(Suffix:='$R',
					Timeout:=T#10MS,
					RxTimeout=>bRxTimeout, StringReceived=>bStringReceived,
					ReceivedString:=sReceivedString255,
					Rxbuffer:=RxBufferPcCom);
UNTIL bStringReceived OR bRxTimeout
END_REPEAT;*)

(*IF bStringReceived THEN
	iState:=1;
END_IF*)

IF nReceivedBytes>0 THEN
	FOR iInd:=0 TO 255 DO
		baReceivedBytes[iInd]:=0;
	END_FOR
	IF (GVL.iSelectedProductType<8) THEN // Ha 6379XX termék
		FOR iInd:=0 TO 26 DO
			baReceivedBytes[iInd]:=RxBufferPcCom.Buffer[iInd];
		END_FOR
	ELSE // Ha 521950 vagy 7459XX termék: 1 karakterrel kevesebb
		FOR iInd:=0 TO 25 DO
			baReceivedBytes[iInd]:=RxBufferPcCom.Buffer[iInd];
		END_FOR
	END_IF
	sReceivedString255:=BYTEARR_TO_MAXSTRING(baReceivedBytes);
	IF LEFT(sReceivedString255,5)='ERROR' THEN
		sReceivedString255:='ERROR';
	END_IF
	nReceivedStringLength:=LEN(sReceivedString255);
	IF nReceivedStringLength>20 THEN
		iState:=1;
	END_IF
	nReceivedBytes:=0;
END_IF

(*ZebraReceiveString(
	Prefix:='',
	Suffix:='',
	Timeout:=T#1S,
	Reset:=bReset,
	StringReceived=>bStringReceived,
	Busy=>bBusy,
	Error=>cetError,
	RxTimeout=>bRxTimeout,
	ReceivedString:=sReceivedString,
	Rxbuffer:=RxBufferPcCom);*)

IF iState=0 AND (bStartSend=TRUE OR bSendBusy=TRUE) THEN
	IF bStartSend=TRUE THEN
//		sStringToSend:=sStartScanning;
		sReceivedString255:='';
		nReceivedStringLength:=0;
		bReadReady:=FALSE;
		GVL.bMarkingOK:=FALSE;
		GVL.iMarkingQ:=0;
		bStart:=TRUE;
	END_IF
(*	IF NOT bKeyence THEN
		ZebraSendData(
			pSendData:=ADR(baStartScanning),
			Length:=6,
			Busy=>bSendBusy,
			Error=>eSendError,
			TXbuffer:=TxBufferPcCom);
	ELSE
		ZebraSendData(
			pSendData:=ADR(baStartScanningKeyence),
			Length:=4,
			Busy=>bSendBusy,
			Error=>eSendError,
			TXbuffer:=TxBufferPcCom);
	END_IF*)
	ClearComBuffer(Buffer:=RxBufferPcCom);
	nReceivedBytes:=0;
	ZebraSendData(
		pSendData:=ADR(baStartScanningKeyence),
		Length:=4,
		Busy=>bSendBusy,
		Error=>eSendError,
		TXbuffer:=TxBufferPcCom);
	bStartSend:=FALSE;
END_IF;

IF bTimeOut=TRUE THEN
	bStart:=FALSE;
	bReadReady:=TRUE;
END_IF

(*IF bStartSend=TRUE OR bSendBusy=TRUE THEN
	IF bStartSend=TRUE THEN
		sStringToSend:=sStartScanning;
	END_IF
	ZebraSendString(
		SendString:=sStringToSend,
		Busy=>bSendBusy,
		Error=>eSendError,
		TXbuffer:=TxBufferPcCom);
	bStartSend:=FALSE;
END_IF;*)

IF iState>0 THEN
	CASE iState OF
		1:	// Időpont beolvasása
			bStartGetTime:=TRUE;
			iState:=2;
		2:	// Várakozás a busy jelre
			IF bGetTimeBusy=TRUE THEN
				iState:=3;
			END_IF
		3:	// Várakozás az időpont beolvasás befejeztére
			IF bGetTimeBusy=FALSE THEN
				bStartGetTime:=FALSE;
				iState:=4;
			END_IF
		4:	// Időpont beolvasás sikerességének vizsgálata
			IF bGetTimeError=FALSE THEN
				iState:=5;
			ELSE
				iState:=100;
			END_IF
		5:	// Szövegek előállítása (pl. a rendszeridőből)
			IF sReceivedString255<>'$04Ð' THEN
				iState:=6;
			END_IF
		6:	// Szövegek előállítása (pl. a rendszeridőből)
			sYear:=WORD_TO_STRING(tstDateTime.wYear);
			sMonth:=WORD_TO_STRING(tstDateTime.wMonth);
			IF tstDateTime.wMonth<10 THEN
				sMonth:=CONCAT('0',sMonth);
			END_IF;
			sDay:=WORD_TO_STRING(tstDateTime.wDay);
			IF tstDateTime.wDay<10 THEN
				sDay:=CONCAT('0',sDay);
			END_IF;
			sExpectedString:=CONCAT('#',
							 CONCAT(sYear,
							 CONCAT(sMonth,sDay)));
			IF (GVL.iSelectedProductType<8) THEN // Ha 6379XX termék
				sTypeCode:=TO_STRING(GVL.iSelectedProductType);
				sExpectedString:=CONCAT('25268941000000A##',
									CONCAT(sTypeCode,sExpectedString));
			ELSIF (GVL.iSelectedProductType>8) THEN // Ha 7459XX termék
				CASE GVL.iSelectedProductType OF
					9, 10: sTypeCode:='0'; //745900 és 745910
					11, 12: sTypeCode:='1'; //745905 és 745915
					13, 14: sTypeCode:='2'; //745906 és 745916
					15, 16: sTypeCode:='3'; //745907 és 745917
				END_CASE
				IF LEFT(GVL.saProductTypes[GVL.iSelectedProductType],5)='74590' THEN
					sExpectedString:=CONCAT('2529534000000A##',
									CONCAT(sTypeCode,sExpectedString));
				ELSE
					sExpectedString:=CONCAT('2529594000000A##',
									CONCAT(sTypeCode,sExpectedString));
				END_IF;
			ELSE
				sExpectedString:=CONCAT('2526894000000A##0',sExpectedString);
			END_IF
			GVL.bMarkingOK:=(sExpectedString=sReceivedString255); // '$04Ð'
			IF GVL.bMarkingOK=TRUE THEN
				GVL.iMarkingQ:=1;
			ELSE	
				GVL.iMarkingQ:=2;
			END_IF
			bReadReady:=TRUE;
			bStart:=FALSE;
			iState:=0;
	END_CASE;
END_IF

Timer(
		IN:=bStart,
		PT:=tTimeOut,
		Q=>bTimeOut,
		ET=>tElapsedTime);
		
GetTime(
		NETID:='',
		START:=bStartGetTime,
		TMOUT:=T#1S,
		BUSY=>bGetTimeBusy,
		ERR=>bGetTimeError,
		ERRID=>nGetTimeError,
		TIMESTR=>tstDateTime
		);

END_PROGRAM

// ---- POUs/PISTI/Components/LOGGING.TcPOU
PROGRAM LOGGING
VAR
	
	// Idő lekérdezése
	GetTime: NT_GetTime;
	bStartGetTime: BOOL;
	bGetTimeBusy: BOOL;
	bGetTimeError: BOOL;
	nGetTimeError: UDINT;
	tstDateTime: TIMESTRUCT;
	dtDateTime: DT;
	
	// Stringek előállítása a logolnivalóhoz
	sLogFilePath: STRING;
	sYear: STRING;
	wWeekOfTheYear: WORD;
	sWeekOfTheYear: STRING;
	sDateTime: STRING;
	sProductType: STRING := '637900';
	sHeaderLine: STRING(255) :=
		'Datum;Zeitpunkt;Produkt;Ref Temp [C];R-Pt1000 [Ohm];Pt1000 Q;R-NTC [Ohm];NTC Q;Zeitkonstant [s];Isolation;Belastungstest Pt1000;DMC Prüfung;Qualifizierung$R$N';
	sHeaderLine2: STRING(255) :=
		'Datum;Zeitpunkt;Produkt;Ref Temp [C];R-Pt1000 [Ohm];Pt1000 Q;R-NTC [Ohm];NTC Q;R-NTC2 [Ohm];NTC2 Q;Zeitkonstant [s];Isolation;Belastungstest Pt1000;DMC Prüfung;Qualifizierung$R$N';
	sTemp: STRING;
	sPTRes: STRING;
	sPtOK: STRING;
	sNTCRes: STRING;
	sNTC2Res: STRING;
	sNTCOK: STRING;
	sNTC2OK: STRING;
	sTimeConst: STRING;
	sIsolOK: STRING;
	sShockOK: STRING;
	sMarkingOK: STRING;
	sQualOK: STRING;
	sLogLine: STRING(255);
	sInfoToLog: STRING(255);
	
	// Fájl infó lekérdezése
	GetFileInfo: fb_EnumFindFileEntry;
	bGetFileInfoExecute: BOOL;
	bGetFileInfoBusy: BOOL;
	bGetFileInfoError: BOOL;
	nGetFileInfoError: UDINT;
	bGetFileInfoEOE: BOOL;
	stLogFile: ST_FindFileEntry;
	
	// Fájl pointer pozíció lekérdezése
//	GetFilePointerPosition: fb_FileTell;	
//	bStartGetPos: BOOL;
//	bGetPosBusy: BOOL;
//	bGetPosError: BOOL;
//	nGetPosError: UDINT;
//	nFilePointerPosition: DINT;
	
	// Fájlnyitás
	bLogOpenExecute: BOOL := FALSE;
	LogOpen: fb_FileOpen;
	nLogOpenMode: DWORD;
	bLogOpenBusy: BOOL;
	bLogOpenError: BOOL;
	nLogOpenError: UDINT;
	hLogFile: UINT;
	
	// Fájlírás
	LogPutStr: fb_FilePuts;
	bLogPutStrExecute: BOOL;
	bLogPutStrBusy: BOOL;
	bLogPutStrError: BOOL;
	nLogPutStrError: UDINT;
	
	// Fájlzárás
	LogClose: fb_FileClose;
	bLogCloseExecute: BOOL;
	bLogCloseBusy: BOOL;
	bLogCloseError: BOOL;
	nLogCloseError: UDINT;
	
	// Könyvtár létrehozása
	CreateDir: fb_CreateDir;	
	sDirectoryName: T_MaxString;
	bCreateDirExecute: BOOL;
	bCreateDirBusy: BOOL;
	bCreateDirError: BOOL;
	nCreateDirError: UDINT;
END_VAR
VAR_INPUT
	iState: INT := 0;
	s_InCommand: STRING := '';
	iProductType: INT :=0;
END_VAR
VAR_OUTPUT
	n_OutErrId: UINT;
END_VAR

IF iState=0 THEN
	IF s_InCommand='LOGOLAS' THEN
		iState:=1;
	ELSE
		s_InCommand:='';
	END_IF
ELSE
	CASE iState OF
		1:	// Időpont beolvasása
			bStartGetTime:=TRUE;
			iState:=2;
		2:	// Várakozás a busy jelre
			IF bGetTimeBusy=TRUE THEN
				iState:=3;
			END_IF
		3:	// Várakozás az időpont beolvasás befejeztére
			IF bGetTimeBusy=FALSE THEN
				bStartGetTime:=FALSE;
				iState:=4;
			END_IF
		4:	// Időpont beolvasás sikerességének vizsgálata
			IF bGetTimeError=FALSE THEN
				iState:=5;
			ELSE
				n_OutErrId:=313;
			END_IF
		5:	// Szövegek előállítása (pl. a rendszeridőből)
			sYear:=WORD_TO_STRING(tstDateTime.wYear);
			dtDateTime:=SYSTEMTIME_TO_DT(tstDateTime);
			wWeekOfTheYear:=F_GetWeekOfTheYear(dtDateTime);
			// Legyen kétszámjegyű a hetek száma:
			IF wWeekOfTheYear<10 THEN
				sWeekOfTheYear:=CONCAT('0',WORD_TO_STRING(wWeekOfTheYear));
			ELSE
				sWeekOfTheYear:=WORD_TO_STRING(wWeekOfTheYear);
			END_IF
			IF GVL.iSelectedProductType<8 THEN
				sLogFilePath:=	CONCAT(CONCAT(CONCAT('C:\Log\',sYear),CONCAT('\','637_KW')),
							CONCAT(sWeekOfTheYear,'.csv'));
			ELSIF GVL.iSelectedProductType>8 THEN
				sLogFilePath:=	CONCAT(CONCAT(CONCAT('C:\Log\',sYear),CONCAT('\','745_KW')),
							CONCAT(sWeekOfTheYear,'.csv'));
			END_IF				
			sDateTime:=CONCAT(DELETE(REPLACE(SYSTEMTIME_TO_STRING(tstDateTime),';',1,11),4,20),';');
			IF GVL.iCurrentProductType=0 THEN
				sProductType:=CONCAT(GVL.saProductTypes[GVL.iSelectedProductType],';');
			ELSE
				IF GVL.iSelectedProductType<8 THEN				
					sProductType:=CONCAT(GVL.saProductTypeNames[GVL.iCurrentProductType],';');
				ELSIF GVL.iSelectedProductType>8 THEN
					sProductType:=CONCAT(GVL.saProductTypeNames745[GVL.iCurrentProductType],';');
				END_IF
			END_IF
			sTemp:=REAL_TO_STRING2(GVL.rTemp,2);
			sTemp:=REPLACE(sTemp,',',1,FIND(sTemp,'.'));
			sTemp:=CONCAT(sTemp,';');
//			sTemp:=CONCAT(REAL_TO_STRING2(GVL.rTemp,2),';');
			sPTRes:=REAL_TO_STRING2(GVL.rPtRes,1);
			sPTRes:=REPLACE(sPTRes,',',1,FIND(sPTRes,'.'));
			sPTRes:=CONCAT(sPTRes,';');
//			sPTRes:=CONCAT(REAL_TO_STRING2(GVL.rPtRes,1),';');
			IF GVL.iPTResQ=0 THEN
				sPtOK:='-;';
			ELSIF GVL.iPTResQ=1 THEN
				sPtOK:='i.O.;';
			ELSE
				sPtOK:='n.i.O.;';				
			END_IF
			sNTCRes:=REAL_TO_STRING2(GVL.rNTCRes,0);
			sNTCRes:=REPLACE(sNTCRes,',',1,FIND(sNTCRes,'.'));
			sNTCRes:=CONCAT(sNTCRes,';');
			sNTC2Res:=REAL_TO_STRING2(GVL.rNTCRes2,0);
			sNTC2Res:=REPLACE(sNTC2Res,',',1,FIND(sNTC2Res,'.'));
			sNTC2Res:=CONCAT(sNTC2Res,';');
//			sNTCRes:=CONCAT(REAL_TO_STRING2(GVL.rNTCRes,0),';');
			IF GVL.iNTCResQ=0 THEN
				sNTCOK:='-;';
			ELSIF GVL.iNTCResQ=1 THEN
				sNTCOK:='i.O.;';
			ELSE
				sNTCOK:='n.i.O.;';				
			END_IF
			IF GVL.iNTC2ResQ=0 THEN
				sNTC2OK:='-;';
			ELSIF GVL.iNTC2ResQ=1 THEN
				sNTC2OK:='i.O.;';
			ELSE
				sNTC2OK:='n.i.O.;';				
			END_IF
			IF GVL.iTimeConstQ=0 THEN
				sTimeConst:='-;';
			ELSIF GVL.iTimeConstQ=1 THEN
				sTimeConst:=REAL_TO_STRING2(GVL.rTimeConst,2);
				sTimeConst:=REPLACE(sTimeConst,',',1,FIND(sTimeConst,'.'));
				sTimeConst:=CONCAT(sTimeConst,';');
//				sTimeConst:=CONCAT(REAL_TO_STRING2(GVL.rTimeConst,2),';');
			ELSE
				sTimeConst:='n.i.O.;';
			END_IF		
			IF GVL.iIsolQ=0 THEN
				sIsolOK:='-;';
			ELSIF GVL.iIsolQ=1 THEN
				sIsolOK:='i.O.;';
			ELSE
				sIsolOK:='n.i.O.;';				
			END_IF
			IF GVL.iShockQ=0 THEN
				sShockOK:='-;';
			ELSIF GVL.iShockQ=1 THEN
				sShockOK:='i.O.;';
			ELSE
				sShockOK:='n.i.O.;';				
			END_IF
			IF GVL.iMarkingQ=0 THEN
				sMarkingOK:='-;';
			ELSIF GVL.iMarkingQ=1 THEN
				sMarkingOK:='i.O.;';
			ELSE
				sMarkingOK:='n.i.O.;';				
			END_IF
(*			IF GVL.bPTResOK=TRUE AND GVL.bNTCResOK=TRUE
				AND GVL.bTimeConstOK=TRUE AND GVL.bIsolOK=TRUE
				AND (GVL.bShockOK=TRUE OR GVL.iCurrentProductType<0)
				AND GVL.bMarkingOK=TRUE THEN*)
			IF GVL.bProductOK=TRUE THEN
				sQualOK:='i.O.$N';
//				sQualOK:='i.O.$R$N';
			ELSE
				sQualOK:='n.i.O.$N';				
//				sQualOK:='n.i.O.$R$N';				
			END_IF
			IF GVL.iSelectedProductType<8 THEN
				sLogLine:=	CONCAT(sDateTime,
							CONCAT(sProductType,
							CONCAT(sTemp,
							CONCAT(sPTRes,
							CONCAT(sPtOK,
							CONCAT(sNTCRes,
							CONCAT(sNTCOK,
							CONCAT(sTimeConst,
							CONCAT(sIsolOK,
							CONCAT(sShockOK,
							CONCAT(sMarkingOK,sQualOK)))))))))));
			ELSE
				sLogLine:=	CONCAT(sDateTime,
							CONCAT(sProductType,
							CONCAT(sTemp,
							CONCAT(sPTRes,
							CONCAT(sPtOK,
							CONCAT(sNTCRes,
							CONCAT(sNTCOK,
							CONCAT(sNTC2Res,
							CONCAT(sNTC2OK,
							CONCAT(sTimeConst,
							CONCAT(sIsolOK,
							CONCAT(sShockOK,
							CONCAT(sMarkingOK,sQualOK)))))))))))));
			END_IF;
			iState:=6;
		6:	// Log fájl megnyitásának kezdeményezése
			bLogOpenExecute:=TRUE;
			nLogOpenMode:=FOPEN_MODETEXT OR FOPEN_MODEAPPEND;
			iState:=7;
		7:	// Várakozás a busy jelre
			IF bLogOpenBusy=TRUE THEN
				iState:=8;
			END_IF
		8:	// Várakozás a fájlnyitás befejeztére
			IF bLogOpenBusy=FALSE THEN
				bLogOpenExecute:=FALSE;
				iState:=9;
			END_IF
		9:	// Fájlnyitás sikerességének vizsgálata
			IF bLogOpenError=FALSE THEN
				iState:=10;
			ELSE
				iState:=101;
			END_IF
		// File méret lekérdezése
		// Ebből állapítható meg, hogy van-e már benne fejléc.
		10:	// File infó lekérdezésének indítása
			bGetFileInfoExecute:=TRUE;
			iState:=11;
		11:	// Várakozás a busy jelre
			IF bGetFileInfoBusy=TRUE THEN
				iState:=12;
			END_IF
		12:	// Várakozás az infólekérdezés befejeztére
			IF bGetFileInfoBusy=FALSE THEN
				bGetFileInfoExecute:=FALSE;
				iState:=13;
			END_IF
		13:	// Infólekérdezés sikerességének vizsgálata
			IF bGetFileInfoError=FALSE AND bGetFileInfoEOE=FALSE THEN
				iState:=14;
			ELSE
				n_OutErrId:=312;
			END_IF
		14:	// Ha most keletkezett a fájl, akkor fejlécet is írunk bele
			IF stLogFile.fileSize.dwLowPart>0
				OR stLogFile.fileSize.dwHighPart>0 THEN
				sInfoToLog:=sLogLine;
			ELSE
				IF GVL.iSelectedProductType<8 THEN
					sInfoToLog:=CONCAT(sHeaderLine,sLogLine);
				ELSE
					sInfoToLog:=CONCAT(sHeaderLine2,sLogLine);
				END_IF
			END_IF
			iState:=15;
		15:	// Log fájlba írás kezdeményezése
			bLogPutStrExecute:=TRUE;
			iState:=16;
		16:	// Várakozás a busy jelre
			IF bLogPutStrBusy=TRUE THEN
				iState:=17;
			END_IF
		17:	// Várakozás a fájlírás befejeztére
			IF bLogPutStrBusy=FALSE THEN
				bLogPutStrExecute:=FALSE;
				iState:=18;
			END_IF
		18:	// Fájlírás sikerességének vizsgálata
			IF bLogPutStrError=FALSE THEN
				iState:=19;
			ELSE
				n_OutErrId:=314;
			END_IF
		19:	// Log fájl zárásának kezdeményezése
			bLogCloseExecute:=TRUE;
			iState:=20;
		20:	// Várakozás a busy jelre
			IF bLogCloseBusy=TRUE THEN
				iState:=21;
			END_IF
		21:	// Várakozás a fájlzárás befejeztére
			IF bLogCloseBusy=FALSE THEN
				bLogCloseExecute:=FALSE;
				iState:=22;
			END_IF
		22:	// Fájlzárás sikerességének vizsgálata
			IF bLogCloseError=FALSE THEN
				iState:=0;
				s_InCommand:='';
				n_OutErrId:=0;
			ELSE
				n_OutErrId:=315;
			END_IF
		40:	// Könyvtár létrehozásának kezdeményezése
			sDirectoryName:=CONCAT('C:\Log\',sYear);
			bCreateDirExecute:=TRUE;
			iState:=41;
		41:	// Várakozás a busy jelre
			IF bCreateDirBusy=TRUE THEN
				iState:=42;
			END_IF
		42:	// Várakozás a fájlnyitás befejeztére
			IF bCreateDirBusy=FALSE THEN
				bCreateDirExecute:=FALSE;
				iState:=43;
			END_IF
		43:	// Fájlnyitás sikerességének vizsgálata
			IF bCreateDirError=FALSE THEN
				iState:=6;
			ELSE
				n_OutErrId:=311;
			END_IF
		101: // Sikertelen fájl létrehozás esetén új könyvtár létrehozása
			IF nLogOpenError=16#70C THEN
				iState:=40;
			ELSE
				n_OutErrId:=311;
			END_IF
	END_CASE
END_IF

LogOpen(
		sNetId:='',
		sPathName:=sLogFilePath,
		nMode:=nLogOpenMode,
		ePath:=PATH_GENERIC,
		bExecute:=bLogOpenExecute,
		tTimeout:=T#5S,
		bBusy=>bLogOpenBusy,
		bError=>bLogOpenError,
		nErrId=>nLogOpenError,
		hFile=>hLogFile
		);
		
LogPutStr(
		sNetId:='',
		hFile:=hLogFile,
		sLine:=sInfoToLog,
		bExecute:=bLogPutStrExecute,
		tTimeout:=T#1S,
		bBusy=>bLogPutStrBusy,
		bError=>bLogPutStrError,
		nErrId=>nLogPutStrError);
		
LogClose(
		sNetId:='',
		hFile:=hLogFile,
		bExecute:=bLogCloseExecute,
		tTimeout:=T#5S,
		bBusy=>bLogCloseBusy,
		bError=>bLogCloseError,
		nErrId=>nLogCloseError
		);
		
GetTime(
		NETID:='',
		START:=bStartGetTime,
		TMOUT:=T#1S,
		BUSY=>bGetTimeBusy,
		ERR=>bGetTimeError,
		ERRID=>nGetTimeError,
		TIMESTR=>tstDateTime
		);
		
//GetFilePointerPosition(
//		sNetId:='',
//		hFile:=hLogFile,
//		bExecute:=bStartGetPos,
//		tTimeout:=T#1S,
//		bBusy=>bGetPosBusy,
//		bError=>bGetPosError,
//		nErrId=>nGetPosError,
//		nSeekPos=>nFilePointerPosition
//		);

GetFileInfo(
		sNetId:='',
		sPathName:=sLogFilePath,
		eCmd:=eEnumCmd_First,
		bExecute:=bGetFileInfoExecute,
		tTimeout:=T#1S,
		bBusy=>bGetFileInfoBusy,
		bError=>bGetFileInfoError,
		nErrId=>nGetFileInfoError,
		bEOE=>bGetFileInfoEOE,
		stFindFile=>stLogFile);

CreateDir(
		sNetId:='',
		sPathName:=sDirectoryName,
		ePath:=PATH_GENERIC,
		bExecute:=bCreateDirExecute,
		tTimeout:=T#1S,
		bBusy=>bCreateDirBusy,
		bError=>bCreateDirError,
		nErrId=>nCreateDirError);

END_PROGRAM

// ---- POUs/PISTI/Helpers/REAL_TO_STRING2.TcPOU
FUNCTION REAL_TO_STRING2 : string
VAR_INPUT
	rIn: LREAL;
	nDigits: BYTE;
END_VAR
VAR
	nMult: DINT := 1;
	nI: BYTE;
END_VAR

FOR nI:=1 TO nDigits DO
	nMult:=nMult*10;
END_FOR
REAL_TO_STRING2:=LREAL_TO_STRING(DINT_TO_LREAL(LREAL_TO_DINT(rIn*nMult))/nMult);

END_FUNCTION

// ---- POUs/JOZSI/Components/HEGESZTESUTMERES.TcPOU
PROGRAM HEGESZTESUTMERES
VAR
	ulDistanceTreshold: ULINT := 141232;
	bMitStromSetting: BOOL;
	bMitStromRestore: BOOL;
//	bAutomaticWeldingStop4: BOOL;
//	bAutomaticWeldingStop5: BOOL;
//	nWeldingStopDistance4: DINT := 320;
//	nWeldingStopDistance5: DINT := 320;
	nMaxWeldingDistance: DINT := 0;
	nWeldingDeformation1: ULINT;
	nWeldingDeformation2: ULINT;
	nWeldingDeformation3: ULINT;
	nWeldingDeformation4: ULINT;
	nWeldingDeformation5: ULINT;
	nWeldingNum: UINT;
	nDistances: ARRAY[0..3000] OF DINT;
	nTimePoints: ARRAY[0..3000] OF DINT;
	sDistance: STRING(4);
	sTimePoint: STRING(4);
	Timer: TON;
	Timer2: TON;
	bStart: BOOL:=FALSE;
	tMaxTime: TIME := T#3.1S;
	tDelayTime: TIME;
	bTimePassed: BOOL;
	tElapsedTime: TIME;
	nI: UINT;
	
	// Idő lekérdezése
	GetTime: NT_GetTime;
	bStartGetTime: BOOL;
	bGetTimeBusy: BOOL;
	bGetTimeError: BOOL;
	nGetTimeError: UDINT;
	tstDateTime: TIMESTRUCT;
	dtDateTime: DT;
	
	// Fájlnyitás
	bLogOpenExecute: BOOL := FALSE;
	LogOpen: fb_FileOpen;
	nLogOpenMode: DWORD;
	bLogOpenBusy: BOOL;
	bLogOpenError: BOOL;
	nLogOpenError: UDINT;
	hLogFile: UINT;
	
	// Fájlírás
	LogPutStr: fb_FilePuts;
	bLogPutStrExecute: BOOL;
	bLogPutStrBusy: BOOL;
	bLogPutStrError: BOOL;
	nLogPutStrError: UDINT;
	LogWriteStr: fb_FileWrite;
//	saLogInfos: ARRAY[0..2002] OF STRING(11);
	saLogInfos: ARRAY[0..3002] OF STRING(10);
	bLogWriteExecute: BOOL;
	bLogWriteBusy: BOOL;
	bLogWriteError: BOOL;
	nLogWriteError: UDINT;
	cbLogWriteLen: UDINT;
	
	// Fájlzárás
	LogClose: fb_FileClose;
	bLogCloseExecute: BOOL;
	bLogCloseBusy: BOOL;
	bLogCloseError: BOOL;
	nLogCloseError: UDINT;
	
	
	sLogFilePath: T_MaxString;
//	sFolder: T_MaxString:='S:\Zoli\637\';
	sFolder: T_MaxString:='C:\Log\';
	sInfoToLog: T_MaxString;
//	sHeader1: STRING(11) := ' Idö [ms] ;';
//	sHeader2: STRING(11) := ' Táv [um]$R$N';
	sHeader1: STRING(10) := ' Idö [ms];';
	sHeader2: STRING(10) := ' Táv [um]$N';
	sDateTime: STRING(255);
	bError: BOOL := FALSE;
	bStart2: BOOL;
	tDelayTime2: TIME;
	bTimePassed2: BOOL;
	tElapsedTime2: TIME;
	tDelay: TIME;
END_VAR
VAR_INPUT
	iState: INT := 1;	
	bHegesztoMitStromOut AT %Q*: BOOL := FALSE;
END_VAR


VAR CONSTANT
	nAlarmFillColor: DWORD := 16#FF0000;
	nNormalFillColor: DWORD := 16#FFFFFF;
END_VAR

IF iState<>0 THEN
	CASE iState OF
		1:	// Indítójelre várás, majd időzítés indítása
			IF ((HEGESZTOK.nHegesztoNum=1) OR (HEGESZTOK.nHegesztoNum=2)
				OR (HEGESZTOK.nHegesztoNum=3) OR (HEGESZTOK.nHegesztoNum=4)
				OR (HEGESZTOK.nHegesztoNum=5)) AND (HEGESZTOK.bHegesztoStart=TRUE) THEN
				bMitStromSetting:=HEGESZTOK.bHegesztoMitStromOut; // Megjegyezzük az eredeti
				nWeldingNum:=HEGESZTOK.nHegesztoNum;	// árambeállítást
				IF (nWeldingNum=1) AND (GVL.bAutomaticWeldingStop1=TRUE) // Ha automata hegesztés leállítás van,
					OR (nWeldingNum=2) AND (GVL.bAutomaticWeldingStop2=TRUE) // akkor be is kapcsoljuk
					OR (nWeldingNum=3) AND (GVL.bAutomaticWeldingStop3=TRUE) // akkor be is kapcsoljuk
					OR (nWeldingNum=4) AND (GVL.bAutomaticWeldingStop4=TRUE) // akkor be is kapcsoljuk
					OR (nWeldingNum=5) AND (GVL.bAutomaticWeldingStop5=TRUE) THEN // akkor be is kapcsoljuk
					HEGESZTOK.bHegesztoMitStromOut:=TRUE;	// automatikusan az áramot.
				END_IF
				FOR nI:=0 TO 3000 DO
					nDistances[nI]:=0;
				END_FOR
				bStart:=TRUE;	// Ez a mérés időtartamának kezdete
				tDelay:=T#0s;
				tDelayTime:=tMaxTime;	// tMaxTime-ig mérünk
				nI:=0;
				nMaxWeldingDistance:=0;
				saLogInfos[0]:=sHeader1;	// A log file első sora
				saLogInfos[1]:=sHeader2;
//				saLogInfos[0]:=' Idö [ms];';	// A log file első sora
//				saLogInfos[1]:=' Táv [um]$N';
				iState:=2;				
			END_IF
		2:	// Mért pont felvétele; Relatív elmozdulás mikronban
			nTimePoints[nI]:=TIME_TO_DINT(tElapsedTime);	// Mérés pillanata
			IF (nI=0) THEN	// Az első mért távolság legyen nulla távolság/deformáció
				CASE nWeldingNum OF
					1, 2, 3: ulDistanceTreshold:=HEGESZTOK.ulHegeszto1Utmero;
					4, 5: ulDistanceTreshold:=HEGESZTOK.ulHegeszto2Utmero;
				END_CASE				
				CASE nWeldingNum OF
					1: ulDistanceTreshold:=HEGESZTOK.ulHegeszto1Utmero;
						GVL.ulWeldingStartDistance1:=HEGESZTOK.ulHegeszto1Utmero;
					2: ulDistanceTreshold:=HEGESZTOK.ulHegeszto1Utmero;
						GVL.ulWeldingStartDistance2:=HEGESZTOK.ulHegeszto1Utmero;
					3: ulDistanceTreshold:=HEGESZTOK.ulHegeszto1Utmero;
						GVL.ulWeldingStartDistance3:=HEGESZTOK.ulHegeszto1Utmero;
					4: ulDistanceTreshold:=HEGESZTOK.ulHegeszto2Utmero;
						GVL.ulWeldingStartDistance4:=HEGESZTOK.ulHegeszto2Utmero;
					5: ulDistanceTreshold:=HEGESZTOK.ulHegeszto2Utmero;
						GVL.ulWeldingStartDistance5:=HEGESZTOK.ulHegeszto2Utmero;
				END_CASE				
			END_IF
			// Mért távolság/deformáció mikronban:
			CASE nWeldingNum OF
				1, 2, 3: 
				nDistances[nI]:=REAL_TO_DINT(ULINT_TO_REAL(ulDistanceTreshold-HEGESZTOK.ulHegeszto1Utmero)*0.368);
				4, 5:
				nDistances[nI]:=REAL_TO_DINT(ULINT_TO_REAL(ulDistanceTreshold-HEGESZTOK.ulHegeszto2Utmero)*0.368);
			END_CASE				
			nMaxWeldingDistance:=MAX(nDistances[nI],nMaxWeldingDistance); // Az eddigi legnagyobb távolság/deformáció
			// 4 karakteres mérési időpont szövegmező előállítása, a kezdő 0-k helyett szóközök
			IF nTimePoints[nI]<10 THEN
				sTimePoint:=CONCAT('   ',DINT_TO_STRING(nTimePoints[nI]));
			ELSIF nTimePoints[nI]<100 THEN
				sTimePoint:=CONCAT('  ',DINT_TO_STRING(nTimePoints[nI]));
			ELSIF nTimePoints[nI]<1000 THEN
				sTimePoint:=CONCAT(' ',DINT_TO_STRING(nTimePoints[nI]));
			ELSE
				sTimePoint:=DINT_TO_STRING(nTimePoints[nI]);
			END_IF
			// 4 karakteres mért távolság/deformáció szövegmezőjének előállítása,
			// a kezdő 0-k helyett szóközök
			IF nDistances[nI]<10 THEN
				sDistance:=CONCAT('   ',DINT_TO_STRING(nDistances[nI]));
			ELSIF nDistances[nI]<100 THEN
				sDistance:=CONCAT('  ',DINT_TO_STRING(nDistances[nI]));
			ELSIF nDistances[nI]<1000 THEN
				sDistance:=CONCAT(' ',DINT_TO_STRING(nDistances[nI]));
			ELSE
				sDistance:=DINT_TO_STRING(nDistances[nI]);
			END_IF
			IF (nI>1000)	// 1000 ms után kapcsolja be a hegesztő az áramot, innentől
				// kell mérni a hegesztési deformációt
				// Ha 1. hegesztés és autostop,
				AND ((GVL.bAutomaticWeldingStop1=TRUE) AND (nWeldingNum=1)
				AND (nDistances[nI]-nDistances[1001]>=GVL.nWeldingStopDistance1)
				// vagy ha 2. hegesztés és autostop,
				OR (GVL.bAutomaticWeldingStop2=TRUE) AND (nWeldingNum=2)
				AND (nDistances[nI]-nDistances[1001]>=GVL.nWeldingStopDistance2)	
				// vagy ha 3. hegesztés és autostop,
				OR (GVL.bAutomaticWeldingStop3=TRUE) AND (nWeldingNum=3)
				AND (nDistances[nI]-nDistances[1001]>=GVL.nWeldingStopDistance3)	
				// vagy ha 4. hegesztés és autostop,
				OR (GVL.bAutomaticWeldingStop4=TRUE) AND (nWeldingNum=4)
				AND (nDistances[nI]-nDistances[401]>=GVL.nWeldingStopDistance4)	
				// vagy ha 5. hegesztés és autostop,
				OR (GVL.bAutomaticWeldingStop5=TRUE) AND (nWeldingNum=5)
				AND (nDistances[nI]-nDistances[401]>=GVL.nWeldingStopDistance5)) THEN
				// akkor a kívánt deformációnál kapcsolja ki az áramot!
				HEGESZTOK.bHegesztoMitStromOut:=FALSE;
			END_IF
			// nI. mérés log sora:
			saLogInfos[nI+2]:=CONCAT(sTimePoint,
							CONCAT(';',
//							CONCAT(sDistance,'$R$N')));
							CONCAT(sDistance,'$N')));
			// Ha betelt a log tömb vagy letelt az 1,5 másodperc, akkor vége a mérésnek,
			IF (nI>2999) OR (tElapsedTime>T#3S) OR (HEGESZTOK.nHegesztoNum=0) THEN // Ha visszahúzódik a hegesztőfej, akkor nincs értelme tovább várni.
//				cbLogWriteLen:=(nI+2)*12; // A mentendő tömb mérete
				cbLogWriteLen:=(nI+2)*11; // A mentendő tömb mérete
				// Hegesztési deformáció kiszámítása
				CASE nWeldingNum OF
					1: GVL.nWeldingDeformation1:=nMaxWeldingDistance-nDistances[1001];
					2: GVL.nWeldingDeformation2:=nMaxWeldingDistance-nDistances[1001];
					3: GVL.nWeldingDeformation3:=nMaxWeldingDistance-nDistances[1001];
					4: GVL.nWeldingDeformation4:=nMaxWeldingDistance-nDistances[401];
					5: GVL.nWeldingDeformation5:=nMaxWeldingDistance-nDistances[401];
				END_CASE
				iState:=3;
			// egyébként a következő mérési pont jön
			ELSE
				nI:=nI+1;
			END_IF;
		3:	// Mérés leállítása
			bStart:=FALSE;
			IF GVL.bWeldingLog=TRUE THEN
				iState:=4;
			ELSE
				iState:=20;
			END_IF;
		4:	// Időpont beolvasása log file-hoz
			bStartGetTime:=TRUE;
			iState:=5;
		5:	// Várakozás a busy jelre
			IF bGetTimeBusy=TRUE THEN
				iState:=6;
			END_IF
		6:	// Várakozás az időpont beolvasás befejeztére
			IF bGetTimeBusy=FALSE THEN
				bStartGetTime:=FALSE;
				iState:=7;
			END_IF
		7:	// Időpont beolvasás sikerességének vizsgálata
			IF bGetTimeError=FALSE THEN
				iState:=8;
			ELSE
				iState:=100;
			END_IF
		8:	// Fájlnév előállítása, fájlnyitás kezdeményezése
			sDateTime:=REPLACE(REPLACE(REPLACE(DELETE(SYSTEMTIME_TO_STRING(tstDateTime),4,20),'-',1,11),'.',1,14),'.',1,17);
			sLogFilePath:=	CONCAT(sFolder,
							CONCAT(sDateTime,'.csv'));
			bLogOpenExecute:=TRUE;
			nLogOpenMode:=FOPEN_MODETEXT OR FOPEN_MODEWRITE;
			iState:=9;
		9:	// Várakozás a busy jelre
			IF bLogOpenBusy=TRUE THEN
				iState:=10;
			END_IF
		10:	// Várakozás a fájlnyitás befejeztére
			IF bLogOpenBusy=FALSE THEN
				bLogOpenExecute:=FALSE;
				iState:=11;
			END_IF
		11:	// Fájlnyitás sikerességének vizsgálata
			IF bLogOpenError=FALSE THEN
				iState:=12;
			ELSE
				iState:=101;
			END_IF
		12:	// Log fájlba írás kezdeményezése
			bLogWriteExecute:=TRUE;
			iState:=13;
		13:	// Várakozás a busy jelre
			IF bLogWriteBusy=TRUE THEN
				iState:=14;
			END_IF
		14:	// Várakozás a fájlírás befejeztére
			IF bLogWriteBusy=FALSE THEN
				bLogWriteExecute:=FALSE;
				iState:=15;
			END_IF
		15:	// Fájlírás sikerességének vizsgálata
			IF bLogWriteError=FALSE THEN
				iState:=16;
			ELSE
				iState:=103;
			END_IF
		16:	// Log fájl zárásának kezdeményezése
			bLogCloseExecute:=TRUE;
			iState:=17;
		17:	// Várakozás a busy jelre
			IF bLogCloseBusy=TRUE THEN
				iState:=18;
			END_IF
		18:	// Várakozás a fájlzárás befejeztére
			IF bLogCloseBusy=FALSE THEN
				bLogCloseExecute:=FALSE;
				iState:=19;
			END_IF
		19:	// Fájlzárás sikerességének vizsgálata
			IF bLogCloseError=FALSE THEN
				iState:=20;
			ELSE
				iState:=104;
			END_IF
		20: // Várakozás a hegesztő program végére
			IF (HEGESZTOK.nHegesztoNum=0) THEN
				iState:=1;
				// Visszakapcsoljuk az eredeti árambeállítást
				HEGESZTOK.bHegesztoMitStromOut:=bMitStromSetting;
			END_IF
	END_CASE
	bError:=(iState>=100);
END_IF

Timer(
		IN:=bStart,
		PT:=tDelayTime,
		Q=>bTimePassed,
		ET=>tElapsedTime);
		
LogOpen(
		sNetId:='',
		sPathName:=sLogFilePath,
		nMode:=nLogOpenMode,
		ePath:=PATH_GENERIC,
		bExecute:=bLogOpenExecute,
		tTimeout:=T#5S,
		bBusy=>bLogOpenBusy,
		bError=>bLogOpenError,
		nErrId=>nLogOpenError,
		hFile=>hLogFile
		);
		
LogPutStr(
		sNetId:='',
		hFile:=hLogFile,
		sLine:=sInfoToLog,
		bExecute:=bLogPutStrExecute,
		tTimeout:=T#1S,
		bBusy=>bLogPutStrBusy,
		bError=>bLogPutStrError,
		nErrId=>nLogPutStrError);
		
LogWriteStr(
		sNetId:='',
		hFile:=hLogFile,
		pWriteBuff:=ADR(saLogInfos),
		cbWriteLen:=cbLogWriteLen,
		bExecute:=bLogWriteExecute,
		tTimeout:=T#1S,
		bBusy=>bLogWriteBusy,
		bError=>bLogWriteError,
		nErrId=>nLogWriteError,
		cbWrite=>);

LogClose(
		sNetId:='',
		hFile:=hLogFile,
		bExecute:=bLogCloseExecute,
		tTimeout:=T#5S,
		bBusy=>bLogCloseBusy,
		bError=>bLogCloseError,
		nErrId=>nLogCloseError
		);

GetTime(
		NETID:='',
		START:=bStartGetTime,
		TMOUT:=T#1S,
		BUSY=>bGetTimeBusy,
		ERR=>bGetTimeError,
		ERRID=>nGetTimeError,
		TIMESTR=>tstDateTime
		);

// Az alábbi kóddal azt az időt mértük, ami az áram kikacsolásának
// szoftverből indítása és a visszajelzés szoftverbe érkezése között eltelt.
// Ennek ideje 13 ms volt.
(*  
IF (bStart2=FALSE) AND (HEGESZTOK.bHegesztoMitStromOut=FALSE)
	AND (HEGESZTOK.bHegesztoMitStromIn=TRUE) THEN
	bStart2:=TRUE;
	tDelayTime2:=T#1H;
	tDelay:=T#0S;
END_IF

IF (bStart2=TRUE) AND (HEGESZTOK.bHegesztoMitStromOut=FALSE)
	AND (HEGESZTOK.bHegesztoMitStromIn=FALSE) THEN
	bStart2:=FALSE;
	tDelay:=tElapsedTime2;
END_IF
		
Timer2(
		IN:=bStart2,
		PT:=tDelayTime2,
		Q=>bTimePassed2,
		ET=>tElapsedTime2);
*)

END_PROGRAM

// ---- POUs/JOZSI/Components/HEGESZTOFEJTISZTITAS.TcPOU
PROGRAM HEGESZTOFEJTISZTITAS
VAR
	iState: INT := 0;
	iCount: INT;
	iMaxCount: INT := 10;
	lrPosition: LREAL := -751; //JOZSITENGELY.lrSardisajatPosition1;
	WAIT: TON;
	bIdoIndul: BOOL;
	bIdoLejart: BOOL := FALSE;
	tDelay: TIME := T#250ms;
END_VAR

IF iState<>0 THEN
	CASE iState OF
		1:	// Inicializálás
			GVL.bJOZSITENGELYReserved:=TRUE;
			iCount:=0;
			iState:=2;
			bIdoIndul:=FALSE;
			lrPosition:=GVL.lrCsiszoloPosition2;
			JOZSITENGELY.lrJozsiPosition:=lrPosition;
			JOZSITENGELY.sJozsiAxisCommand:='MOVE';
			iState:=2;
		2:	// Kezdő pozíció felvétele
			IF JOZSITENGELY.sJozsiAxisCommand='' THEN
				iState:=3;
			END_IF;
		3: // 1. hegesztőfej le
			HEGESZTOK.nHegesztoNum:=GVL.nHegFejTisztProgram-1;
			iState:=4;
		4:	// Késleltetés indítása
			bIdoIndul:=TRUE;
			iState:=5;
		5:	// Várakozás a késleltetés lejártára
			IF bIdoLejart=TRUE THEN
				bIdoIndul:=FALSE;
				iState:=6;
			END_IF
		6:	// Ha lent van a fej, akkor egy mozgás és számol egyet 
			IF (HEGESZTOK.ulHegeszto1Utmero<142500) THEN
				IF lrPosition=GVL.lrCsiszoloPosition1 THEN
					lrPosition:=GVL.lrCsiszoloPosition2;
				ELSIF lrPosition=GVL.lrCsiszoloPosition2 THEN
					lrPosition:=GVL.lrCsiszoloPosition1;
				END_IF
				GVL.bHegesztofejTisztitas:=TRUE;
				JOZSITENGELY.lrJozsiPosition:=lrPosition;
				JOZSITENGELY.sJozsiAxisCommand:='MOVE';
				iCount:=iCount+1;
				iState:=7;
			END_IF;
		7:	// Ha még nem mozgott eleget, akkor vissza a mozgásra, különben kilépés
			IF (JOZSITENGELY.sJozsiAxisCommand='') THEN
				IF iCount<2*GVL.nHegFejTisztCiklusok THEN
					iState:=4;
				ELSE
					iState:=8;
					GVL.bHegesztofejTisztitas:=FALSE;
				END_IF
			END_IF
		8:	// Hegesztőfej fel
//			IF (GVL.bHegeszto1BalLent=TRUE) THEN
				HEGESZTOK.nHegesztoNum:=0;
				iState:=9;			
//			END_IF
		9:	// Ha a hegesztőfej fent van, akkor következő lépés
			IF (GVL.bHegeszto1BalFent=TRUE)
				AND (GVL.bHegeszto1JobbFent=TRUE) THEN
				iState:=100;
			END_IF
		100: // Szervizboxhoz
			JOZSITENGELY.lrJozsiPosition:=GVL.lrNTCSzervizbox;
			JOZSITENGELY.sJozsiAxisCommand:='MOVE';
			iState:=101;
		101: IF JOZSITENGELY.sJozsiAxisCommand='' THEN
				iState:=0;
				GVL.bJOZSITENGELYReserved:=FALSE;
			END_IF;
	END_CASE
END_IF
WAIT(IN:=bIdoIndul,PT:=tDelay,Q=>bIdoLejart,ET=>);

END_PROGRAM

// ---- POUs/JOZSI/Components/KAMERA.TcPOU
PROGRAM KAMERA
VAR
	iState: INT;
	bVizsgalatKesz: BOOL := FALSE;
	FB_Idozites: TON;
	FB_TriggerPulse: TP;
	
	// Kamera szoftver megnyitása
	FB_Start_IVNav: NT_StartProcess;
	bStartIVNav: BOOL;
	bIVNavBusy: BOOL;
	bIVNavErr: BOOL;
	nIVNavErr: UDINT;
	iState2: INT;

	bStartIdozites: BOOL;
	bIdozitesLejart: BOOL;
	bTriggerPulse: BOOL;
END_VAR

CASE iState OF
	0:
		IF GVL.bKameraTrigger=TRUE THEN
			bVizsgalatKesz:=FALSE;
			bStartIdozites:=TRUE;
			iState:=2;
		END_IF
	1:
		IF GVL.bKameraBusy=TRUE THEN
			iState:=2;
		END_IF
	2:
(*		IF GVL.bKameraBusy=FALSE THEN *)
		IF bIdozitesLejart=TRUE THEN
			bStartIdozites:=FALSE;
			GVL.bKameraTrigger:=FALSE;
			bVizsgalatKesz:=TRUE;
			iState:=0;
		END_IF
END_CASE

CASE iState2 OF
	0:	// Várakozás parancsra
		IF (bStartIVNav=TRUE) THEN
			iState2:=1;
		END_IF
	1:
		IF (bIVNavBusy=TRUE) THEN
			iState2:=2;
		END_IF
	2:
		IF (bIVNavBusy=FALSE) THEN
			bStartIVNav:=FALSE;
			iState2:=0;
		END_IF
END_CASE

FB_Idozites(IN:=bStartIdozites,
			PT:=T#100MS,
			Q => bIdozitesLejart);

// Kamera saját szoftverének indítása
FB_Start_IVNav(
					NETID:='',
					PATHSTR:='C:\Program Files\KEYENCE\IV-Navigator\IV-Navigator.exe',
					DIRNAME:='C:\Program Files\KEYENCE\IV-Navigator\',
					COMNDLINE:='',
					START:=bStartIVNav,
					TMOUT:=T#30S,
					BUSY => bIVNavBusy,
					ERR => bIVNavErr,
					ERRID => nIVNavErr
					);

FB_TriggerPulse(
				IN:=GVL.bPtKameraTrigger,
				PT:=T#150MS,
				Q => bTriggerPulse);
GVL.bPtKameraTrigger:=bTriggerPulse;

END_PROGRAM

// ---- POUs/GENERAL/Components/BARCODE_SCANNER.TcPOU
PROGRAM BARCODE_SCANNER
VAR
	iState: INT := 0;
	iInd: DINT;
	iInd2: INT;

	TxBufferPcCom: COMbuffer;
	RxBufferPcCom: COMbuffer;
	fbPCComCtrl: SerialLineControlADS;
	bConnect: BOOL := TRUE;
	stSerialCfgZebra: ComSerialConfig := (ComPort := 5, DTR := COMDTRCTRL_T.DTR_CTRL_DISABLE, RTS := COMRTSCTRL_T.RTS_CTRL_ENABLE);
	bPortOpened: BOOL;
	bPcComCtrlError: BOOL;
	ePcComCtrlErrorId: UDINT;
	bPCComCtrlBusy: BOOL;
	uiTxBufferCount: UDINT;
	uiRxBufferCount: UDINT;
	baReceivedBytes: ARRAY[0..255] OF BYTE;
	ZebraReceiveBytes: ReceiveByte;
	ClearComBuffer: ClearComBuffer;
	sReceivedString255: T_MaxString;
END_VAR

fbPCComCtrl(
	Connect:=bConnect,
	SerialCfg:=stSerialCfgZebra,
	NetId:='',
	Timeout:=T#2S,
	PortOpened=>bPortOpened,
	Error=>bPCComCtrlError,
	ErrorId=>ePCComCtrlErrorId,
	Busy=>bPCComCtrlBusy,
	TxBufCount=>uiTxBufferCount,
	RxBufCount=>uiRxBufferCount,
	TxBuffer:=TxBufferPcCom,
	RxBuffer:=RxBufferPcCom);


REPEAT
	ZebraReceiveBytes(Rxbuffer:=RxBufferPcCom);
UNTIL NOT ZebraReceiveBytes.ByteReceived
END_REPEAT;

GVL.LogButtonsDis:=GVL.LoginEnabled OR GVL.AddDeleteEnabled;
GVL.AddDelButtonDis:=GVL.LoginEnabled OR GVL.AddDeleteEnabled;

IF RxBufferPcCom.RdIdx > 0 THEN
	FOR iInd:=0 TO 255 DO
		baReceivedBytes[iInd]:=0;
	END_FOR
	FOR iInd:= 0 TO RxBufferPcCom.RdIdx-1 DO
		baReceivedBytes[iInd]:=RxBufferPcCom.Buffer[iInd];
	END_FOR
	sReceivedString255:='';
	sReceivedString255:=BYTEARR_TO_MAXSTRING(baReceivedBytes);
	ClearComBuffer(Buffer:=RxBufferPcCom);
	iState:=1;
END_IF

IF NOT GVL.LoginEnabled THEN
	GVL.UserNotFound:=FALSE;	
END_IF

IF GVL.Biztos THEN
	IF GVL.AddDeleteEnabled THEN
		GVL.UserDelete:=TRUE;
	END_IF
	GVL.Biztos:=FALSE;
END_IF

IF GVL.Logout_Button THEN
	GVL.UserActual := GVL.Users[0];
	GVL.Logout_Button:=FALSE;
	GVL.AddDeleteEnabled:=FALSE;
END_IF

IF GVL.AddDeleteEnabled THEN
	IF GVL.UserID_Temp <> GVL.UserID_Elozo THEN
		GVL.UserTemp:=GVL.Users[GVL.UserID_Temp];
		GVL.UserTemp.UserID:=GVL.UserID_Temp;
		GVL.UserID_Elozo:=GVL.UserID_Temp;
	END_IF
ELSE
	GVL.UserID_Temp:=0;
	GVL.UserID_Elozo:=GVL.UserID_Temp;
	GVL.UserTemp:=GVL.Users[GVL.UserID_Temp];
END_IF

IF GVL.UserModify THEN
	IF GVL.UserTemp.UserID <> 0 THEN
		GVL.Users[GVL.UserID_Temp]:=GVL.UserTemp;
		GVL.Users[GVL.UserID_Temp].UserExist:=TRUE;
		GVL.bStart_WrPer:=TRUE;
	END_IF
	GVL.UserModify:=FALSE;
END_IF

IF GVL.UserDelete THEN
	IF GVL.UserTemp.UserID <> 0 AND GVL.UserTemp.UserID <> GVL.UserActual.UserID THEN
		GVL.Users[GVL.UserID_Temp].UserLevel:=0;
		GVL.Users[GVL.UserID_Temp].UserName:='';
		GVL.Users[GVL.UserID_Temp].UserNumber:='';
		GVL.Users[GVL.UserID_Temp].UserExist:=FALSE;
		GVL.Users[GVL.UserID_Temp].UserID:=0;
		GVL.UserID_Temp:=0;
		GVL.UserID_Elozo:=GVL.UserID_Temp;
		GVL.UserTemp:=GVL.Users[GVL.UserID_Temp];
	END_IF
	GVL.UserDelete:=FALSE;
END_IF

IF iState>0 THEN
	CASE iState OF
		1:	
			IF GVL.LoginEnabled THEN
				GVL.UserNotFound := FALSE;
				IF GVL.UserActual.UserNumber <> sReceivedString255 THEN
					FOR iInd2 := 0 TO 99 DO
						IF sReceivedString255 = GVL.Users[iInd2].UserNumber THEN
							GVL.UserActual := GVL.Users[iInd2];
							GVL.UserNotFound := FALSE;
							EXIT;							
						END_IF
						GVL.UserNotFound := TRUE;
					END_FOR					
				END_IF
				IF NOT GVL.UserNotFound THEN
					GVL.LoginEnabled := FALSE;
				END_IF
				iState:=0;
			ELSE
				iState:=10;
			END_IF
		10:	
			IF GVL.AddDeleteEnabled THEN
				IF GVL.UserTemp.UserID>0 THEN
					GVL.UserTemp.UserNumber:=sReceivedString255;
				END_IF
				iState:=0;
			ELSE
				iState:=20;
			END_IF
		20:
			iState:=0;
	END_CASE;
END_IF

END_PROGRAM

// ---- CheckDivDInt.TcPOU
// Implicitly generated code : DO NOT EDIT
FUNCTION CheckDivDInt : DINT
VAR_INPUT
	divisor:DINT;
END_VAR

// Implicitly generated code : Only an Implementation suggestion
{noflow}
IF divisor = 0 THEN
	CheckDivDInt:=1;
ELSE
	CheckDivDInt:=divisor;
END_IF;
{flow}

END_FUNCTION

// ---- CheckDivLInt.TcPOU
// Implicitly generated code : DO NOT EDIT
FUNCTION CheckDivLInt : LINT
VAR_INPUT
	divisor:LINT;
END_VAR

// Implicitly generated code : Only an Implementation suggestion
{noflow}
IF divisor = 0 THEN
	CheckDivLInt:=1;
ELSE
	CheckDivLInt:=divisor;
END_IF;
{flow}

END_FUNCTION

// ---- CheckDivLReal.TcPOU
// Implicitly generated code : DO NOT EDIT
FUNCTION CheckDivLReal : LREAL
VAR_INPUT
	divisor:LREAL;
END_VAR

// Implicitly generated code : Only an Implementation suggestion
{noflow}
IF divisor = 0 THEN
	CheckDivLReal:=1;
ELSE
	CheckDivLReal:=divisor;
END_IF;
{flow}

END_FUNCTION

// ---- CheckDivReal.TcPOU
// Implicitly generated code : DO NOT EDIT
FUNCTION CheckDivReal : REAL
VAR_INPUT
	divisor:REAL;
END_VAR

// Implicitly generated code : Only an Implementation suggestion
{noflow}
IF divisor = 0 THEN
	CheckDivReal:=1;
ELSE
	CheckDivReal:=divisor;
END_IF;
{flow}

END_FUNCTION

// ---- CheckLRangeSigned.TcPOU
// Implicitly generated code : DO NOT EDIT
FUNCTION CheckLRangeSigned : LINT
VAR_INPUT
	value, lower, upper: LINT;
END_VAR

// Implicitly generated code : Only an Implementation suggestion
{noflow}
IF (value < lower) THEN
	CheckLRangeSigned := lower;
ELSIF(value > upper) THEN
	CheckLRangeSigned := upper;
ELSE
	CheckLRangeSigned := value;
END_IF

{flow}

END_FUNCTION

// ---- CheckLRangeUnsigned.TcPOU
// Implicitly generated code : DO NOT EDIT
FUNCTION CheckLRangeUnsigned : ULINT
VAR_INPUT
	value, lower, upper: ULINT;
END_VAR

// Implicitly generated code : Only an Implementation suggestion
{noflow}
IF (value < lower) THEN
	CheckLRangeUnsigned := lower;
ELSIF(value > upper) THEN
	CheckLRangeUnsigned := upper;
ELSE
	CheckLRangeUnsigned := value;
END_IF
{flow}

END_FUNCTION

// ---- CheckPointer.TcPOU
// Implicitly generated code : DO NOT EDIT
FUNCTION CheckPointer : POINTER TO BYTE
VAR_INPUT 
	ptToTest : POINTER TO BYTE; // Destination address of the pointer
	iSize : DINT;		        // Size of the type the pointer points to. (e.g: 20 for POINTER TO ARRAY [0..9] OF INT) 
	iGran : DINT;		        // Granularity of the pointer access. This is the size of the biggest non-structured data type in the type the pointer points to. (e.g: 2 for POINTER TO ARRAY [0..9] OF INT)
	bWrite: BOOL;		        // Indicates read or write Access. TRUE = write access.
END_VAR

// No standard way of implementation. Fill your own code here
CheckPointer := ptToTest;
{flow}

END_FUNCTION

// ---- CheckRangeSigned.TcPOU
// Implicitly generated code : DO NOT EDIT
FUNCTION CheckRangeSigned : DINT
VAR_INPUT
	value, lower, upper: DINT;
END_VAR

// Implicitly generated code : Only an Implementation suggestion
{noflow}
IF (value < lower) THEN
	CheckRangeSigned := lower;
ELSIF(value > upper) THEN
	CheckRangeSigned := upper;
ELSE
	CheckRangeSigned := value;
END_IF
{flow}

END_FUNCTION

// ---- CheckRangeUnsigned.TcPOU
// Implicitly generated code : DO NOT EDIT
FUNCTION CheckRangeUnsigned : UDINT
VAR_INPUT
	value, lower, upper: UDINT;
END_VAR

// Implicitly generated code : Only an Implementation suggestion
{noflow}
IF (value < lower) THEN
	CheckRangeUnsigned := lower;
ELSIF(value > upper) THEN
	CheckRangeUnsigned := upper;
ELSE
	CheckRangeUnsigned := value;
END_IF
{flow}

END_FUNCTION

// ---- POUs/CheckBounds.TcPOU
// Implicitly generated code : DO NOT EDIT
FUNCTION CheckBounds : DINT
VAR_INPUT
	index, lower, upper: DINT;
END_VAR

// Implicitly generated code : Only an Implementation suggestion
{noflow}
IF  index < lower THEN
	CheckBounds := lower;
ELSIF  index > upper THEN
	CheckBounds := upper;
ELSE  
	CheckBounds := index;
END_IF
{flow}

END_FUNCTION

// ---- POUs/GENERAL/Components/Robot/ROBOTCOMMAND_OLD.TcPOU
PROGRAM ROBOTCOMMAND_OLD
VAR_INPUT
	bRobotCommOpenEnable : BOOL := FALSE;
	sRobotCommand : STRING := '';
END_VAR
VAR_OUTPUT
	bRobotCommOpen : BOOL := FALSE;
	nRobotErrId: UDINT;
	sRobotResult : STRING := '';
END_VAR
VAR	
//LOCALS
	//Kapcsolat nyitás
	sRobotRemoteHost: STRING := '192.168.1.100';
	bRobotSocketbusy: BOOL;
	bRobotSocketError: BOOL;
	nRobotSocketErrId: UDINT;
	hRobotSocket: T_HSOCKET;
	bRobotSocketOpenEnable: BOOL := FALSE;
	RobotSocketOpen: FB_SocketConnect;
	
	//Küldés
	RobotSocketSend: FB_SocketSend;
	baSendByteArray: ARRAY[0..255] OF BYTE;
	bRobotSocketSendEnable: BOOL := FALSE;
	sLRobotCommand: STRING :='';
	sRobotSendData: STRING;
	uSendByteLen: UDINT := 0;
	bRobotSocketSendbusy: BOOL;
	bRobotSocketSendError: BOOL;
	nRobotSocketSendErrId: UDINT;
	
	//Fogadás
	RobotSocketReceive: FB_SocketReceive;
	baReceivedByteArray: ARRAY[0..255] OF BYTE;
	bRobotSocketReceiveEnable: BOOL := FALSE;
	sRobotReceived: STRING :='';
	nRobotReceivedBytesNum: UDINT;
	bRobotSocketReceivebusy: BOOL;
	bRobotSocketReceiveError: BOOL;
	nRobotSocketReceiveErrId: UDINT;
	
	//Kapcsolat bontás
	bRobotSocketCloseEnable: BOOL := FALSE;
	RobotSocketClose: FB_SocketClose;
END_VAR


IF bRobotCommOpenEnable = TRUE THEN
	//Kommunikáció nyitás
	IF NOT(bRobotCommOpen) THEN
		RobotSocketOpen(
			sSrvNetId:= '', 
			sRemoteHost:= sRobotRemoteHost, 
			nRemotePort:= 2000, 
			bExecute:= bRobotSocketOpenEnable, 
			tTimeout:= T#45S, 
			bBusy=> bRobotSocketbusy, 
			bError=> bRobotSocketError, 
			nErrId=> nRobotSocketErrId, 
			hSocket=> hRobotSocket);
		IF bRobotSocketOpenEnable=TRUE THEN
			IF (NOT(bRobotSocketError) AND NOT(bRobotSocketbusy)) THEN
				bRobotSocketOpenEnable := FALSE;
				bRobotCommOpen:=TRUE;
				MEMSET(ADR(baReceivedByteArray), 0, 256);
				RobotSocketOpen(
					sSrvNetId:= '', 
					sRemoteHost:= sRobotRemoteHost, 
					nRemotePort:= 2000, 
					bExecute:= FALSE, 
					tTimeout:= T#45S, 
					bBusy=> bRobotSocketbusy, 
					bError=> bRobotSocketError, 
					nErrId=> nRobotSocketErrId, 
					hSocket=> hRobotSocket);
			END_IF
		ELSE
			bRobotSocketOpenEnable:=TRUE;
		END_IF
	END_IF
END_IF

IF (sLRobotCommand = '' AND sRobotCommand<>'' AND bRobotCommOpen = TRUE) THEN
	nRobotErrId := 0;
	sLRobotCommand := sRobotCommand;
	sRobotResult := sRobotCommand;
END_IF

//Adatküldés
IF sLRobotCommand<>'' AND bRobotCommOpen=TRUE THEN
	RobotSocketSend(
		sSrvNetId:= '', 
		hSocket:= hRobotSocket, 
		cbLen:= uSendByteLen, 
		pSrc:= ADR(baSendByteArray), 
		bExecute:= bRobotSocketSendEnable, 
		tTimeout:= T#5S, 
		bBusy=> bRobotSocketSendbusy, 
		bError=> bRobotSocketSendError, 
		nErrId=> nRobotSocketSendErrId);
		
	IF bRobotSocketSendEnable=TRUE THEN
		IF NOT(bRobotSocketSendbusy) THEN		
			bRobotSocketSendEnable:=FALSE;
			IF NOT(bRobotSocketSendError) THEN
				sLRobotCommand:='';
				sRobotCommand:='';
			ELSE
				nRobotErrId := nRobotSocketSendErrId;
				sLRobotCommand := '';
				sRobotCommand:='';
			END_IF;
		END_IF;
	ELSE
		sRobotSendData := sLRobotCommand;
		baSendByteArray := MAXSTRING_TO_BYTEARR(sRobotSendData);
		uSendByteLen := INT_TO_UDINT(LEN(sRobotSendData));
		bRobotSocketSendEnable:=TRUE;
	END_IF
END_IF

//Adatfogadás
IF bRobotCommOpen=TRUE THEN
	RobotSocketReceive(
		sSrvNetId:= '', 
		hSocket:= hRobotSocket, 
		cbLen:= 255, 
		pDest:= ADR(baReceivedByteArray), 
		bExecute:= bRobotSocketReceiveEnable, 
		tTimeout:= T#5S, 
		bBusy=> bRobotSocketReceivebusy, 
		bError=> bRobotSocketReceiveError, 
		nErrId=> nRobotSocketReceiveErrId, 
		nRecBytes=> nRobotReceivedBytesNum);
		
	IF bRobotSocketReceiveEnable=TRUE THEN
		IF NOT(bRobotSocketReceivebusy) THEN	
			bRobotSocketReceiveEnable:=FALSE;
			IF NOT(bRobotSocketReceiveError) THEN
				IF nRobotReceivedBytesNum<>0 THEN
					sRobotReceived := BYTEARR_TO_MAXSTRING(baReceivedByteArray);
					MEMSET(ADR(baReceivedByteArray), 0, 256);
					IF sRobotReceived[0] = 16#30 THEN
						sRobotResult := DELETE(sRobotReceived,1,1);
						nRobotErrId:= 0;
					ELSE
						sRobotResult := DELETE(sRobotReceived,1,1);
						nRobotErrId:= 10000;
					END_IF
				END_IF;
			ELSE
				sRobotResult:='';
				nRobotErrId := nRobotSocketReceiveErrId;
			END_IF;
		END_IF;
	ELSE
		nRobotReceivedBytesNum:=0;
		bRobotSocketReceiveEnable := TRUE;
	END_IF;
END_IF

IF bRobotCommOpenEnable = FALSE THEN
	//Kommunikáció bontás
	IF bRobotCommOpen THEN
		RobotSocketClose(
			sSrvNetId:= '', 
			hSocket:= hRobotSocket, 
			bExecute:= bRobotSocketCloseEnable, 
			tTimeout:= T#45S, 
			bBusy=> bRobotSocketbusy, 
			bError=> bRobotSocketError, 
			nErrId=> nRobotSocketErrId);
	IF bRobotSocketCloseEnable=TRUE THEN
			IF (NOT(bRobotSocketError) AND NOT(bRobotSocketError) AND NOT(bRobotSocketbusy)) THEN
				bRobotSocketCloseEnable := FALSE;
				bRobotCommOpen:=FALSE;
				RobotSocketClose(
					sSrvNetId:= '', 
					hSocket:= hRobotSocket, 
					bExecute:= bRobotSocketCloseEnable, 
					tTimeout:= T#45S, 
					bBusy=> bRobotSocketbusy, 
					bError=> bRobotSocketError, 
					nErrId=> nRobotSocketErrId);
			END_IF
		ELSE
			bRobotSocketCloseEnable:=TRUE;
		END_IF
	END_IF
END_IF

END_PROGRAM

// ---- POUs/GENERAL/Components/Robot/ROBOTREMOTE_OLD.TcPOU
PROGRAM ROBOTREMOTE_OLD
VAR_INPUT
	bRobotCommOpenEnable : BOOL := FALSE;
	bRobotCommandSend : BOOL := FALSE;
	sRobotCommand : STRING := '';
	sRobotCommandParam1 : STRING := '';
	sRobotCommandParam2 : STRING := '';
	sRobotCommandParam3 : STRING := '';
	sRobotCommandParam4 : STRING := '';
	sRobotCommandParam5 : STRING := '';
END_VAR
VAR_OUTPUT
	bRobotCommOpen : BOOL := FALSE;
	nRobotErrId: UDINT;
	sRobotResult : STRING := '';
END_VAR
VAR	
//LOCALS
	//RobotComm
	sRobotRemoteHost: STRING := '192.168.1.100';
//	sRobotRemoteHost: STRING := '192.168.1.22';
	bRobotSocketbusy: BOOL;
	bRobotSocketError: BOOL;
	nRobotSocketErrId: UDINT;
	hRobotSocket: T_HSOCKET;
	
	//Kapcsolat nyitás
	bRobotSocketOpenEnable: BOOL := FALSE;
	RobotSocketOpen: FB_SocketConnect;
	
	//Küldés
	bExecuting : BOOL := FALSE;
	bRobotSocketSendEnable: BOOL := FALSE;
	RobotSocketSend: FB_SocketSend;
	sLRobotCommandForResult: STRING :='';
	sLRobotCommand: STRING :='';
	sLRobotParam1: STRING :='';
	sLRobotParam2: STRING :='';
	sLRobotParam3: STRING :='';
	sLRobotParam4: STRING :='';
	sLRobotParam5: STRING :='';
	sRobotSendData: STRING;
	uSendByteLen: UDINT := 0;
	baSendByteArray: ARRAY[0..255] OF BYTE;
	bRobotSocketReceiveEnable: BOOL := FALSE;
	RobotSocketReceive: FB_SocketReceive;
	sRobotReceived: STRING :='';
	nRobotReceivedBytesNum: UDINT;
	baReceivedByteArray: ARRAY[0..255] OF BYTE;
	iTemp : INT := 0;
	
	//Fogadás kiértékelés
	fb_ResultSplitter : fb_SplitRobotResult;
	bIsError : BOOL;
	sErrorOrResult : STRING;
	
	//Kapcsolat bontás
	bRobotSocketCloseEnable: BOOL := FALSE;
	RobotSocketClose: FB_SocketClose;
END_VAR

//Kommunikáció nyitás
IF bRobotCommOpenEnable = TRUE THEN
	IF NOT(bRobotCommOpen) THEN
		RobotSocketOpen(
			sSrvNetId:= '', 
			sRemoteHost:= sRobotRemoteHost, 
			nRemotePort:= 5000, 
//			nRemotePort:= 100, 
			bExecute:= bRobotSocketOpenEnable, 
			tTimeout:= T#45S, 
			bBusy=> bRobotSocketbusy, 
			bError=> bRobotSocketError, 
			nErrId=> nRobotSocketErrId, 
			hSocket=> hRobotSocket);
		IF bRobotSocketOpenEnable=TRUE THEN
			IF (NOT(bRobotSocketError) AND NOT(bRobotSocketError) AND NOT(bRobotSocketbusy)) THEN
				bRobotSocketOpenEnable := FALSE;
				bRobotCommOpen:=TRUE;
				RobotSocketOpen(
					sSrvNetId:= '', 
					sRemoteHost:= sRobotRemoteHost, 
					nRemotePort:= 5000, 
					bExecute:= FALSE, 
					tTimeout:= T#45S, 
					bBusy=> bRobotSocketbusy, 
					bError=> bRobotSocketError, 
					nErrId=> nRobotSocketErrId, 
					hSocket=> hRobotSocket);
			END_IF
		ELSE
			bRobotSocketOpenEnable:=TRUE;
		END_IF
	END_IF
END_IF

IF (NOT(bExecuting) AND (bRobotCommandSend=TRUE) AND bRobotCommOpen) THEN
	nRobotErrId := 0;
	sLRobotCommandForResult := sRobotCommand;
	sLRobotCommand := sRobotCommand;
	sLRobotParam1 := sRobotCommandParam1;
	sLRobotParam2 := sRobotCommandParam2;
	sLRobotParam3 := sRobotCommandParam3;
	sLRobotParam4 := sRobotCommandParam4;
	sLRobotParam5 := sRobotCommandParam5;
END_IF

//Adatküldés
IF sLRobotCommand<>'' THEN
	RobotSocketSend(
		sSrvNetId:= '', 
		hSocket:= hRobotSocket, 
		cbLen:= uSendByteLen, 
		pSrc:= ADR(baSendByteArray), 
		bExecute:= bRobotSocketSendEnable, 
		tTimeout:= T#5S, 
		bBusy=> bRobotSocketbusy, 
		bError=> bRobotSocketError, 
		nErrId=> nRobotSocketErrId);
		
	IF bRobotSocketSendEnable=TRUE THEN
		IF NOT(bRobotSocketbusy) THEN		
			bRobotSocketSendEnable:=FALSE;
			IF NOT(bRobotSocketError) THEN
				sLRobotCommand:='';
				sLRobotCommand := '';
				sLRobotParam1 := '';
				sLRobotParam2 := '';
				sLRobotParam3 := '';
				sLRobotParam4 := '';
				sLRobotParam5 := '';
			ELSE
				nRobotErrId := nRobotSocketErrId;
				bExecuting := FALSE;
				sLRobotCommand := '';
				sLRobotCommand := '';
				sLRobotParam1 := '';
				sLRobotParam2 := '';
				sLRobotParam3 := '';
				sLRobotParam4 := '';
				sLRobotParam5 := '';
			END_IF;
		END_IF;
	ELSE
		sRobotSendData := f_RobotCommandTranslation(sLRobotCommand,sLRobotParam1,sLRobotParam2,sLRobotParam3,sLRobotParam4,sLRobotParam5);
		baSendByteArray := MAXSTRING_TO_BYTEARR(sRobotSendData);
		uSendByteLen := INT_TO_UDINT(LEN(sRobotSendData));
		bRobotSocketSendEnable:=TRUE;
		bExecuting := TRUE;
		bRobotCommandSend := FALSE;
		MEMSET(ADR(baReceivedByteArray), 0, 256);
	END_IF
END_IF

//Adatfogadás
IF bExecuting AND NOT(bRobotSocketSendEnable)  AND bRobotCommOpen THEN
	RobotSocketReceive(
	sSrvNetId:= '', 
	hSocket:= hRobotSocket, 
	cbLen:= 255, 
	pDest:= ADR(baReceivedByteArray), 
	bExecute:= bRobotSocketReceiveEnable, 
	tTimeout:= T#5S, 
	bBusy=> bRobotSocketbusy, 
	bError=> bRobotSocketError, 
	nErrId=> nRobotSocketErrId, 
	nRecBytes=> nRobotReceivedBytesNum);
	
	IF bRobotSocketReceiveEnable=TRUE THEN
		IF NOT(bRobotSocketbusy) THEN	
			bRobotSocketReceiveEnable:=FALSE;
			IF NOT(bRobotSocketError) THEN
				IF nRobotReceivedBytesNum=0 THEN
					bRobotSocketReceiveEnable:=FALSE;
				ELSE
					sRobotReceived := BYTEARR_TO_MAXSTRING(baReceivedByteArray);
					fb_ResultSplitter(sCommand:= sLRobotCommandForResult, sResult:= sRobotReceived, bIsError=> bIsError, sErrorOrResult=> sErrorOrResult);
					IF bIsError THEN
						nRobotErrId:=STRING_TO_UDINT(sErrorOrResult);
						sRobotResult:='';
					ELSE
						nRobotErrId:=0;
						sRobotResult:=sErrorOrResult;
					END_IF
					sRobotCommand := '';
					sRobotCommandParam1 := '';
					sRobotCommandParam2 := '';
					sRobotCommandParam3 := '';
					sRobotCommandParam4 := '';
					sRobotCommandParam5 := '';
					nRobotErrId:= 0;
					bExecuting := FALSE;
				END_IF;
			ELSE
				sRobotCommand := '';
				sRobotCommandParam1 := '';
				sRobotCommandParam2 := '';
				sRobotCommandParam3 := '';
				sRobotCommandParam4 := '';
				sRobotCommandParam5 := '';
				sRobotResult:='';
				nRobotErrId := nRobotSocketErrId;
				bExecuting := FALSE;
			END_IF;
		END_IF;
	ELSE
		nRobotReceivedBytesNum:=0;
		bRobotSocketReceiveEnable := TRUE;
	END_IF;
END_IF

IF bRobotCommOpenEnable = FALSE THEN
	//Kommunikáció bontás
	IF bRobotCommOpen THEN
		RobotSocketClose(
			sSrvNetId:= '', 
			hSocket:= hRobotSocket, 
			bExecute:= bRobotSocketCloseEnable, 
			tTimeout:= T#45S, 
			bBusy=> bRobotSocketbusy, 
			bError=> bRobotSocketError, 
			nErrId=> nRobotSocketErrId);
		IF bRobotSocketCloseEnable=TRUE THEN
				IF (NOT(bRobotSocketError) AND NOT(bRobotSocketError) AND NOT(bRobotSocketbusy)) THEN
					bRobotSocketCloseEnable := FALSE;
					bRobotCommOpen:=FALSE;
					RobotSocketClose(
					sSrvNetId:= '', 
					hSocket:= hRobotSocket, 
					bExecute:= bRobotSocketCloseEnable, 
					tTimeout:= T#45S, 
					bBusy=> bRobotSocketbusy, 
					bError=> bRobotSocketError, 
					nErrId=> nRobotSocketErrId);
				END_IF
		ELSE
			bRobotSocketCloseEnable:=TRUE;
		END_IF
	END_IF
END_IF

END_PROGRAM

// ---- POUs/GENERAL/Helpers/GetResourceFromCommand.TcPOU
FUNCTION GetResourceFromCommand : STRING
VAR_INPUT
	Command: STRING;
END_VAR
VAR
	sReturn : STRING;
END_VAR

sReturn := LEFT ( Command , FIND(Command,'_') - 1);
GetResourceFromCommand := sReturn;

END_FUNCTION

// ---- POUs/GENERAL/Executors/f_E_Robot.TcPOU
FUNCTION f_E_Robot : DINT
VAR_INPUT
	s_Command : STRING := '';
	s_Param1 : STRING := '';
	s_Param2 : STRING := '';
	s_Param3 : STRING := '';
	s_Param4 : STRING := '';
	s_Param5 : STRING := '';
END_VAR
VAR
	s_RobotCommandType : STRING := '';
	b_TypeFound : BOOL := FALSE;
END_VAR

s_RobotCommandType := RIGHT ( s_Command , FIND(s_Command,'_'));
IF ROBOTCOMMAND.sRobotCommand = '' AND ROBOTREMOTE.sRobotCommand = '' THEN
	IF s_RobotCommandType = 'REMOTE' THEN
		RobotProcess.s_InRobotCommand := s_Param1;
		RobotProcess.s_InRobotCommandParam1 := s_Param2;
		RobotProcess.s_InRobotCommandParam2 := s_Param3;
		RobotProcess.s_InRobotCommandParam3 := s_Param4;
		RobotProcess.s_InRobotCommandParam4 := s_Param5;
		b_TypeFound := TRUE;
	END_IF
	IF s_RobotCommandType = 'COMMAND' THEN
		RobotProcess.s_InRobotTCPCommand := s_Param1;
		b_TypeFound := TRUE;
	END_IF
	IF b_TypeFound = FALSE THEN
		f_E_Robot := -101;
	ELSE
		IF RobotProcess.iState = 100 THEN
			f_E_Robot := -200;
		END_IF
	END_IF
ELSE
	f_E_Robot := -100;
END_IF

END_FUNCTION

// ---- POUs/JozsiProcess.TcPOU
PROGRAM JozsiProcess
VAR
	//Futtatáshoz
	bRunning : BOOL := FALSE;
	bIsError : BOOL := FALSE;
	nErrorNum : DINT := 0;
	iPtr : INT := 0;
	sResource : STRING := '';
	bResourceFound : BOOL := FALSE;
	
	//Recepthez
	asActualProgram : ARRAY [0..5,0..199] OF STRING;
	sRecipeName : STRING :='';
END_VAR

IF bRunning=TRUE AND nErrorNum = 0 THEN
		IF (asActualProgram[0,iPtr]) <> '' THEN
			sResource := GetResourceFromCommand(asActualProgram[0,iPtr]);
			IF sResource = 'ROBOT' THEN
				nErrorNum := f_E_Robot(asActualProgram[0,iPtr],asActualProgram[1,iPtr],asActualProgram[2,iPtr],asActualProgram[3,iPtr],asActualProgram[4,iPtr],asActualProgram[5,iPtr]);
			END_IF
			IF nErrorNum <> 0 THEN
				bRunning := FALSE;
			END_IF
		END_IF
//			GVL.sRobotCommand := f_RobotCommandTranslation(asActualProgram[0,iPtr],asActualProgram[1,iPtr],asActualProgram[2,iPtr],asActualProgram[3,iPtr],asActualProgram[4,iPtr],asActualProgram[5,iPtr]);
//			iPtr := iPtr + 1;
//		ELSE
//			bRobotRunning := FALSE;	
//		END_IF
END_IF

END_PROGRAM

// ---- POUs/JOZSI/Components/HEGESZTESUTMERES_1.TcPOU
PROGRAM HEGESZTESUTMERES_1
VAR
	ulDistanceTreshold: ULINT := 141232;
	bMitStromSetting: BOOL;
	bMitStromRestore: BOOL;
//	bAutomaticWeldingStop4: BOOL;
//	bAutomaticWeldingStop5: BOOL;
//	nWeldingStopDistance4: DINT := 320;
//	nWeldingStopDistance5: DINT := 320;
	nMaxWeldingDistance: DINT := 0;
	nWeldingDeformation4: DINT;
	nWeldingDeformation5: DINT;
	nWeldingNum: UINT;
	nDistances: ARRAY[0..2000] OF DINT;
	nTimePoints: ARRAY[0..2000] OF DINT;
	sDistance: STRING(4);
	sTimePoint: STRING(4);
	Timer: TON;
	Timer2: TON;
	bStart: BOOL:=FALSE;
	tMaxTime: TIME := T#1.8S;
	tDelayTime: TIME;
	bTimePassed: BOOL;
	tElapsedTime: TIME;
	nI: UINT;
	
	// Idő lekérdezése
	GetTime: NT_GetTime;
	bStartGetTime: BOOL;
	bGetTimeBusy: BOOL;
	bGetTimeError: BOOL;
	nGetTimeError: UDINT;
	tstDateTime: TIMESTRUCT;
	dtDateTime: DT;
	
	// Fájlnyitás
	bLogOpenExecute: BOOL := FALSE;
	LogOpen: fb_FileOpen;
	nLogOpenMode: DWORD;
	bLogOpenBusy: BOOL;
	bLogOpenError: BOOL;
	nLogOpenError: UDINT;
	hLogFile: UINT;
	
	// Fájlírás
	LogPutStr: fb_FilePuts;
	bLogPutStrExecute: BOOL;
	bLogPutStrBusy: BOOL;
	bLogPutStrError: BOOL;
	nLogPutStrError: UDINT;
	LogWriteStr: fb_FileWrite;
//	saLogInfos: ARRAY[0..2002] OF STRING(11);
	saLogInfos: ARRAY[0..2002] OF STRING(10);
	bLogWriteExecute: BOOL;
	bLogWriteBusy: BOOL;
	bLogWriteError: BOOL;
	nLogWriteError: UDINT;
	cbLogWriteLen: UDINT;
	
	// Fájlzárás
	LogClose: fb_FileClose;
	bLogCloseExecute: BOOL;
	bLogCloseBusy: BOOL;
	bLogCloseError: BOOL;
	nLogCloseError: UDINT;
	
	
	sLogFilePath: T_MaxString;
//	sFolder: T_MaxString:='S:\Zoli\637\';
	sFolder: T_MaxString:='C:\Log\';
	sInfoToLog: T_MaxString;
//	sHeader1: STRING(11) := ' Idö [ms] ;';
//	sHeader2: STRING(11) := ' Táv [um]$R$N';
	sHeader1: STRING(10) := ' Idö [ms];';
	sHeader2: STRING(10) := ' Táv [um]$N';
	sDateTime: STRING(255);
	bError: BOOL := FALSE;
	bStart2: BOOL;
	tDelayTime2: TIME;
	bTimePassed2: BOOL;
	tElapsedTime2: TIME;
	tDelay: TIME;
END_VAR
VAR_INPUT
	iState: INT := 1;	
	bHegesztoMitStromOut AT %Q*: BOOL := FALSE;
END_VAR


VAR CONSTANT
	nAlarmFillColor: DWORD := 16#FF0000;
	nNormalFillColor: DWORD := 16#FFFFFF;
END_VAR

IF iState<>0 THEN
	CASE iState OF
		1:	// Indítójelre várás, majd időzítés indítása
			IF ((HEGESZTOK.nHegesztoNum=4) OR (HEGESZTOK.nHegesztoNum=5)) 
				AND (HEGESZTOK.bHegesztoStart=TRUE) THEN
				bMitStromSetting:=HEGESZTOK.bHegesztoMitStromOut; // Megjegyezzük az eredeti
				nWeldingNum:=HEGESZTOK.nHegesztoNum;	// árambeállítást
				IF (nWeldingNum=4) AND (GVL.bAutomaticWeldingStop4=TRUE) // Ha automata hegesztés leállítás van,
					OR (nWeldingNum=5) AND (GVL.bAutomaticWeldingStop5=TRUE) THEN // akkor be is kapcsoljuk
					HEGESZTOK.bHegesztoMitStromOut:=TRUE;	// automatikusan az áramot.
				END_IF
				bStart:=TRUE;	// Ez a mérés időtartamának kezdete
				tDelay:=T#0s;
				tDelayTime:=tMaxTime;	// tMaxTime-ig mérünk
				nI:=0;
				nMaxWeldingDistance:=0;
				saLogInfos[0]:=sHeader1;	// A log file első sora
				saLogInfos[1]:=sHeader2;
//				saLogInfos[0]:=' Idö [ms];';	// A log file első sora
//				saLogInfos[1]:=' Táv [um]$N';
				iState:=2;				
			END_IF
		2:	// Mért pont felvétele; Relatív elmozdulás mikronban
			nTimePoints[nI]:=TIME_TO_DINT(tElapsedTime);	// Mérés pillanata
			IF (nI=0) THEN	// Az első mért távolság legyen nulla távolság/deformáció
				ulDistanceTreshold:=HEGESZTOK.ulHegeszto2Utmero;
			END_IF
			// Mért távolság/deformáció mikronban:
			nDistances[nI]:=REAL_TO_DINT(ULINT_TO_REAL(ulDistanceTreshold-HEGESZTOK.ulHegeszto2Utmero)*0.368);
			nMaxWeldingDistance:=MAX(nDistances[nI],nMaxWeldingDistance); // Az eddigi legnagyobb távolság/deformáció
			// 4 karakteres mérési időpont szövegmező előállítása, a kezdő 0-k helyett szóközök
			IF nTimePoints[nI]<10 THEN
				sTimePoint:=CONCAT('   ',DINT_TO_STRING(nTimePoints[nI]));
			ELSIF nTimePoints[nI]<100 THEN
				sTimePoint:=CONCAT('  ',DINT_TO_STRING(nTimePoints[nI]));
			ELSIF nTimePoints[nI]<1000 THEN
				sTimePoint:=CONCAT(' ',DINT_TO_STRING(nTimePoints[nI]));
			ELSE
				sTimePoint:=DINT_TO_STRING(nTimePoints[nI]);
			END_IF
			// 4 karakteres mért távolság/deformáció szövegmezőjének előállítása,
			// a kezdő 0-k helyett szóközök
			IF nDistances[nI]<10 THEN
				sDistance:=CONCAT('   ',DINT_TO_STRING(nDistances[nI]));
			ELSIF nDistances[nI]<100 THEN
				sDistance:=CONCAT('  ',DINT_TO_STRING(nDistances[nI]));
			ELSIF nDistances[nI]<1000 THEN
				sDistance:=CONCAT(' ',DINT_TO_STRING(nDistances[nI]));
			ELSE
				sDistance:=DINT_TO_STRING(nDistances[nI]);
			END_IF
			IF (nI>1000)	// 1000 ms után kapcsolja be a hegesztő az áramot, innentől
				// kell mérni a hegesztési deformációt
				// Ha 4. hegesztés és autostop,
				AND ((GVL.bAutomaticWeldingStop4=TRUE) AND (nWeldingNum=4)
				AND (nDistances[nI]-nDistances[401]>=GVL.nWeldingStopDistance4)	
				// vagy ha 5. hegesztés és autostop,
				OR (GVL.bAutomaticWeldingStop5=TRUE) AND (nWeldingNum=5)
				AND (nDistances[nI]-nDistances[401]>=GVL.nWeldingStopDistance5)) THEN
				// akkor a kívánt deformációnál kapcsolja ki az áramot!
				HEGESZTOK.bHegesztoMitStromOut:=FALSE;
			END_IF
			// nI. mérés log sora:
			saLogInfos[nI+2]:=CONCAT(sTimePoint,
							CONCAT(';',
//							CONCAT(sDistance,'$R$N')));
							CONCAT(sDistance,'$N')));
			// Ha betelt a log tömb vagy letelt az 1,5 másodperc, akkor vége a mérésnek,
			IF (nI>1999) OR (tElapsedTime>T#1.5S) THEN
//				cbLogWriteLen:=(nI+2)*12; // A mentendő tömb mérete
				cbLogWriteLen:=(nI+2)*11; // A mentendő tömb mérete
				// Hegesztési deformáció kiszámítása
				IF (nWeldingNum=4) THEN
					nWeldingDeformation4:=nMaxWeldingDistance-nDistances[401];
				ELSIF (nWeldingNum=5) THEN
					nWeldingDeformation5:=nMaxWeldingDistance-nDistances[401];
				END_IF
				iState:=3;
			// egyébként a következő mérési pont jön
			ELSE
				nI:=nI+1;
			END_IF;
		3:	// Mérés leállítása
			bStart:=FALSE;
			iState:=4;
		4:	// Időpont beolvasása log file-hoz
			bStartGetTime:=TRUE;
			iState:=5;
		5:	// Várakozás a busy jelre
			IF bGetTimeBusy=TRUE THEN
				iState:=6;
			END_IF
		6:	// Várakozás az időpont beolvasás befejeztére
			IF bGetTimeBusy=FALSE THEN
				bStartGetTime:=FALSE;
				iState:=7;
			END_IF
		7:	// Időpont beolvasás sikerességének vizsgálata
			IF bGetTimeError=FALSE THEN
				iState:=8;
			ELSE
				iState:=100;
			END_IF
		8:	// Fájlnév előállítása, fájlnyitás kezdeményezése
			sDateTime:=REPLACE(REPLACE(REPLACE(DELETE(SYSTEMTIME_TO_STRING(tstDateTime),4,20),'-',1,11),'.',1,14),'.',1,17);
			sLogFilePath:=	CONCAT(sFolder,
							CONCAT(sDateTime,'.csv'));
			bLogOpenExecute:=TRUE;
			nLogOpenMode:=FOPEN_MODETEXT OR FOPEN_MODEWRITE;
			iState:=9;
		9:	// Várakozás a busy jelre
			IF bLogOpenBusy=TRUE THEN
				iState:=10;
			END_IF
		10:	// Várakozás a fájlnyitás befejeztére
			IF bLogOpenBusy=FALSE THEN
				bLogOpenExecute:=FALSE;
				iState:=11;
			END_IF
		11:	// Fájlnyitás sikerességének vizsgálata
			IF bLogOpenError=FALSE THEN
				iState:=12;
			ELSE
				iState:=101;
			END_IF
		12:	// Log fájlba írás kezdeményezése
			bLogWriteExecute:=TRUE;
			iState:=13;
		13:	// Várakozás a busy jelre
			IF bLogWriteBusy=TRUE THEN
				iState:=14;
			END_IF
		14:	// Várakozás a fájlírás befejeztére
			IF bLogWriteBusy=FALSE THEN
				bLogWriteExecute:=FALSE;
				iState:=15;
			END_IF
		15:	// Fájlírás sikerességének vizsgálata
			IF bLogWriteError=FALSE THEN
				iState:=16;
			ELSE
				iState:=103;
			END_IF
		16:	// Log fájl zárásának kezdeményezése
			bLogCloseExecute:=TRUE;
			iState:=17;
		17:	// Várakozás a busy jelre
			IF bLogCloseBusy=TRUE THEN
				iState:=18;
			END_IF
		18:	// Várakozás a fájlzárás befejeztére
			IF bLogCloseBusy=FALSE THEN
				bLogCloseExecute:=FALSE;
				iState:=19;
			END_IF
		19:	// Fájlzárás sikerességének vizsgálata
			IF bLogCloseError=FALSE THEN
				iState:=20;
			ELSE
				iState:=104;
			END_IF
		20: // Várakozás a hegesztő program végére
			IF (HEGESZTOK.nHegesztoNum=0) THEN
				iState:=1;
				// Visszakapcsoljuk az eredeti árambeállítást
				HEGESZTOK.bHegesztoMitStromOut:=bMitStromSetting;
			END_IF
	END_CASE
	bError:=(iState>=100);
END_IF

Timer(
		IN:=bStart,
		PT:=tDelayTime,
		Q=>bTimePassed,
		ET=>tElapsedTime);
		
LogOpen(
		sNetId:='',
		sPathName:=sLogFilePath,
		nMode:=nLogOpenMode,
		ePath:=PATH_GENERIC,
		bExecute:=bLogOpenExecute,
		tTimeout:=T#5S,
		bBusy=>bLogOpenBusy,
		bError=>bLogOpenError,
		nErrId=>nLogOpenError,
		hFile=>hLogFile
		);
		
LogPutStr(
		sNetId:='',
		hFile:=hLogFile,
		sLine:=sInfoToLog,
		bExecute:=bLogPutStrExecute,
		tTimeout:=T#1S,
		bBusy=>bLogPutStrBusy,
		bError=>bLogPutStrError,
		nErrId=>nLogPutStrError);
		
LogWriteStr(
		sNetId:='',
		hFile:=hLogFile,
		pWriteBuff:=ADR(saLogInfos),
		cbWriteLen:=cbLogWriteLen,
		bExecute:=bLogWriteExecute,
		tTimeout:=T#1S,
		bBusy=>bLogWriteBusy,
		bError=>bLogWriteError,
		nErrId=>nLogWriteError,
		cbWrite=>);

LogClose(
		sNetId:='',
		hFile:=hLogFile,
		bExecute:=bLogCloseExecute,
		tTimeout:=T#5S,
		bBusy=>bLogCloseBusy,
		bError=>bLogCloseError,
		nErrId=>nLogCloseError
		);

GetTime(
		NETID:='',
		START:=bStartGetTime,
		TMOUT:=T#1S,
		BUSY=>bGetTimeBusy,
		ERR=>bGetTimeError,
		ERRID=>nGetTimeError,
		TIMESTR=>tstDateTime
		);

// Az alábbi kóddal azt az időt mértük, ami az áram kikacsolásának
// szoftverből indítása és a visszajelzés szoftverbe érkezése között eltelt.
// Ennek ideje 13 ms volt.
(*  
IF (bStart2=FALSE) AND (HEGESZTOK.bHegesztoMitStromOut=FALSE)
	AND (HEGESZTOK.bHegesztoMitStromIn=TRUE) THEN
	bStart2:=TRUE;
	tDelayTime2:=T#1H;
	tDelay:=T#0S;
END_IF

IF (bStart2=TRUE) AND (HEGESZTOK.bHegesztoMitStromOut=FALSE)
	AND (HEGESZTOK.bHegesztoMitStromIn=FALSE) THEN
	bStart2:=FALSE;
	tDelay:=tElapsedTime2;
END_IF
		
Timer2(
		IN:=bStart2,
		PT:=tDelayTime2,
		Q=>bTimePassed2,
		ET=>tElapsedTime2);
*)

END_PROGRAM

// ---- POUs/JOZSI/Executors/f_E_Tengely.TcPOU
FUNCTION f_E_Tengely : DINT
VAR_INPUT
	s_Command : STRING := '';
	s_Param1 : STRING := '';
	s_Param2 : STRING := '';
	s_Param3 : STRING := '';
	s_Param4 : STRING := '';
	s_Param5 : STRING := '';
END_VAR
VAR
	b_TypeFound : BOOL := FALSE;
END_VAR

IF JOZSITENGELY.sJozsiAxisCommand = '' THEN
	JOZSITENGELY.sJozsiAxisCommand := s_Param1;
	JOZSITENGELY.lrJozsiPosition := STRING_TO_LREAL(s_Param2);
ELSE
	f_E_Tengely := -100;
END_IF

END_FUNCTION

// ---- POUs/PISTI/Components/Laser_old.TcPOU
PROGRAM Laser_old
VAR_INPUT
	s_InCommand : STRING :='';
	s_TypeCode : STRING :='0';	
END_VAR
VAR
	//LaserComm
	sLaserRemoteHost: STRING := '192.168.1.99';
//	sLaserRemoteHost: STRING := '192.168.1.22';
	LaserSocketOpen: FB_SocketConnect;
	bLaserSocketbusy: BOOL;
	bLaserSocketError: BOOL;
	nLaserSocketErrId: UDINT;
	hLaserSocket: T_HSOCKET;
	bLaserSocketOpenEnable: BOOL := FALSE;
	LaserSocketClose: FB_SocketClose;
	bLaserSocketCloseEnable: BOOL := FALSE;
	LaserSocketSend: FB_SocketSend;
	bLaserSocketSendEnable: BOOL := FALSE;
	sLaserSendData: STRING;
	uSendByteLen: UDINT := 0;
	baSendByteArray: ARRAY[0..255] OF BYTE;
	bLaserSocketReceiveEnable: BOOL := FALSE;
	bLaserSocketReceiveRequest: BOOL := FALSE;
	baReceivedByteArray: ARRAY[0..255] OF BYTE;
	sLaserSend: STRING :='';
	sLaserReceived: STRING :='';
	bLaserSendReady: BOOL := TRUE;
	bLaserSendOK: BOOL := FALSE;
	bEvenCycle: BOOL := FALSE;
	LaserSocketReceive: FB_SocketReceive;
	nLaserReceivedBytesNum: UDINT;
	bLogin: BOOL;
END_VAR

